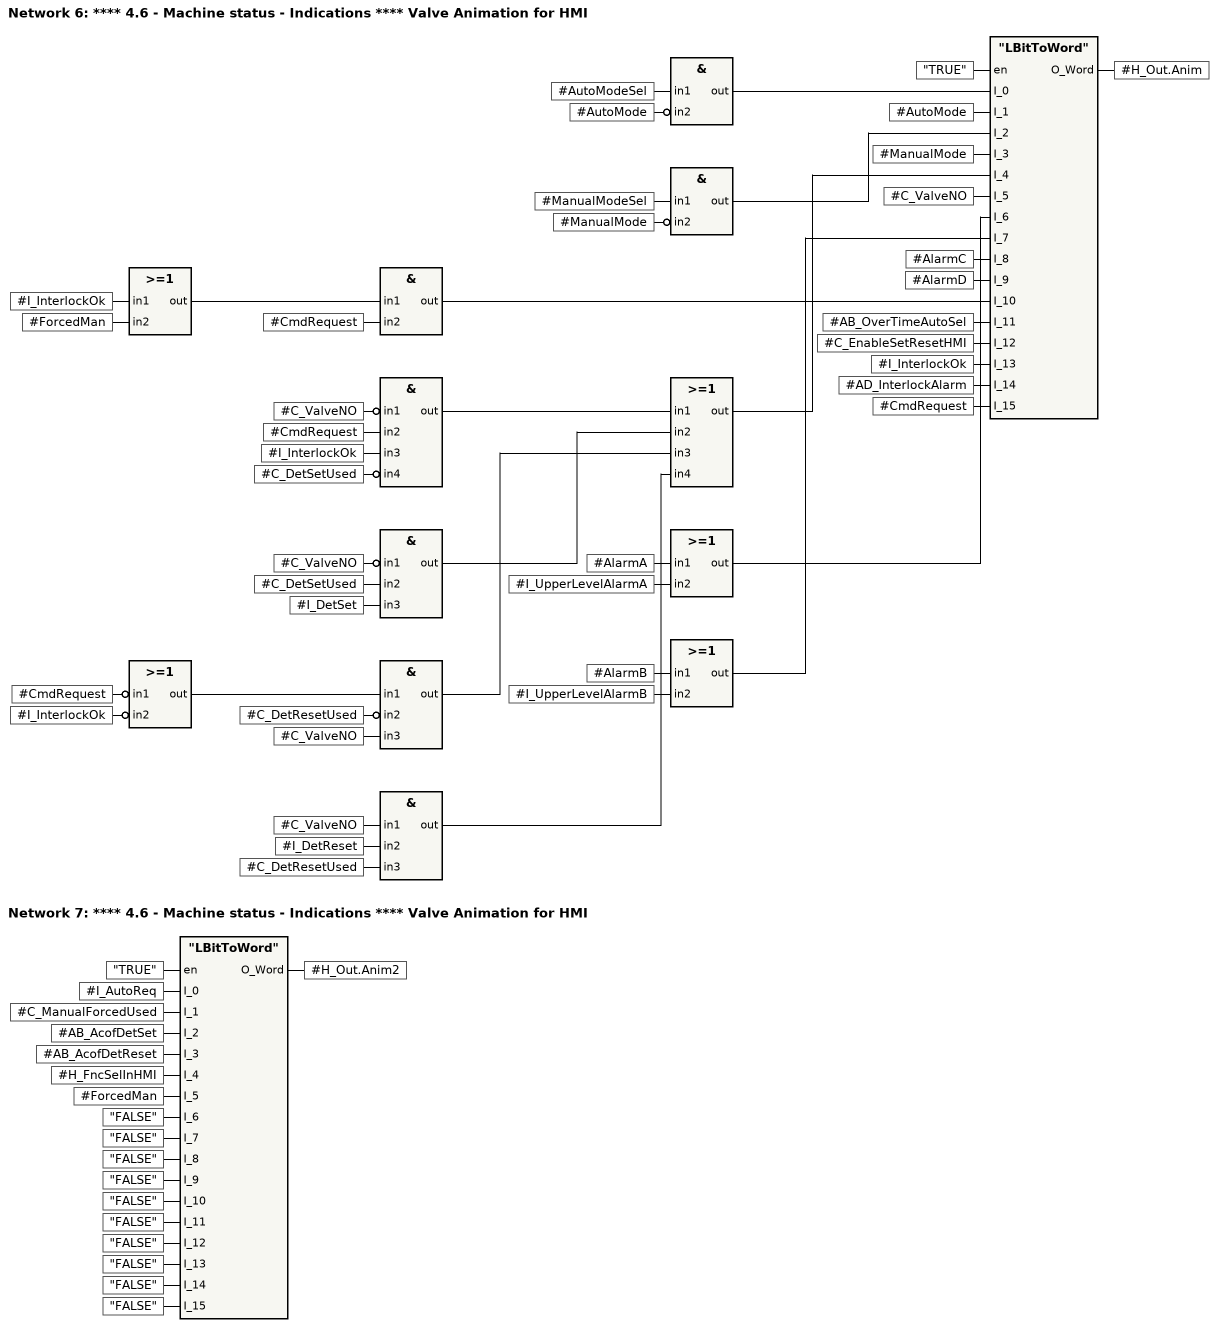
   IF "TRUE" THEN
       "LBitToWord"(I_0 := #AutoModeSel AND NOT #AutoMode,
                    I_1 := #AutoMode,
                    I_2 := #ManualModeSel AND NOT #ManualMode,
                    I_3 := #ManualMode,
                    I_4 := (NOT #C_ValveNO AND #CmdRequest AND #I_InterlockOk AND NOT #C_DetSetUsed) OR (NOT #C_ValveNO AND #C_DetSetUsed AND #I_DetSet) OR ((NOT #CmdRequest OR NOT #I_InterlockOk) AND NOT #C_DetResetUsed AND #C_ValveNO) OR (#C_ValveNO AND #I_DetReset AND #C_DetResetUsed),
                    I_5 := #C_ValveNO,
                    I_6 := #AlarmA OR #I_UpperLevelAlarmA,
                    I_7 := #AlarmB OR #I_UpperLevelAlarmB,
                    I_8 := #AlarmC,
                    I_9 := #AlarmD,
                    I_10 := (#I_InterlockOk OR #ForcedMan) AND #CmdRequest,
                    I_11 := #AB_OverTimeAutoSel,
                    I_12 := #C_EnableSetResetHMI,
                    I_13 := #I_InterlockOk,
                    I_14 := #AD_InterlockAlarm,
                    I_15 := #CmdRequest,
                    O_Word => #H_Out.Anim);
   END_IF;
END_REGION

REGION Network 7: **** 4.6 - Machine status - Indications **** Valve Animation for HMI
   // Valve Animation for HMI
   IF "TRUE" THEN
       "LBitToWord"(I_0 := #I_AutoReq,
                    I_1 := #C_ManualForcedUsed,
                    I_2 := #AB_AcofDetSet,
                    I_3 := #AB_AcofDetReset,
                    I_4 := #H_FncSelInHMI,
                    I_5 := #ForcedMan,
                    I_6 := "FALSE",
                    I_7 := "FALSE",
                    I_8 := "FALSE",
                    I_9 := "FALSE",
                    I_10 := "FALSE",
                    I_11 := "FALSE",
                    I_12 := "FALSE",
                    I_13 := "FALSE",
                    I_14 := "FALSE",
                    I_15 := "FALSE",
                    O_Word => #H_Out.Anim2);
   END_IF;
END_REGION

REGION Network 8: **** 4.6 - Machine status - Indications **** Valve Animation for HMI
   // Valve Animation for HMI
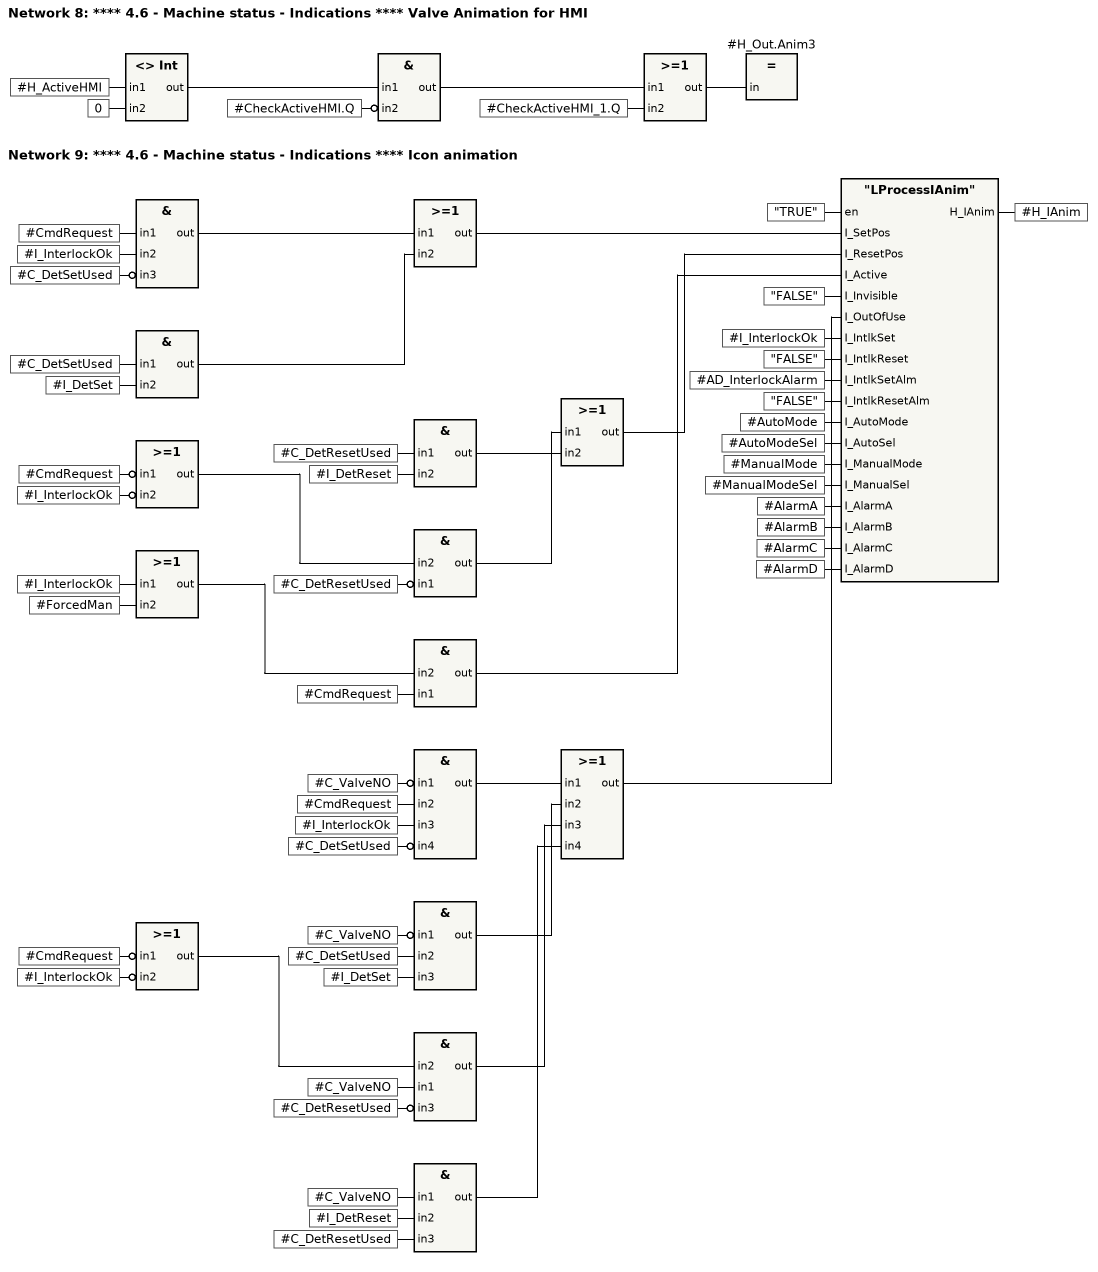
   #H_Out.Anim3 := ((#H_ActiveHMI <> 0) AND NOT #CheckActiveHMI.Q) OR #CheckActiveHMI_1.Q;
END_REGION

REGION Network 9: **** 4.6 - Machine status - Indications **** Icon animation
   // Icon animation
   IF "TRUE" THEN
       "LProcessIAnim"(I_SetPos := (#CmdRequest AND #I_InterlockOk AND NOT #C_DetSetUsed) OR (#C_DetSetUsed AND #I_DetSet),
                       I_ResetPos := ((NOT #CmdRequest OR NOT #I_InterlockOk) AND NOT #C_DetResetUsed) OR (#C_DetResetUsed AND #I_DetReset),
                       I_Active := (#I_InterlockOk OR #ForcedMan) AND #CmdRequest,
                       I_Invisible := "FALSE",
                       I_OutOfUse := (NOT #C_ValveNO AND #CmdRequest AND #I_InterlockOk AND NOT #C_DetSetUsed) OR (NOT #C_ValveNO AND #C_DetSetUsed AND #I_DetSet) OR ((NOT #CmdRequest OR NOT #I_InterlockOk) AND #C_ValveNO AND NOT #C_DetResetUsed) OR (#C_ValveNO AND #I_DetReset AND #C_DetResetUsed),
                       I_IntlkSet := #I_InterlockOk,
                       I_IntlkReset := "FALSE",
                       I_IntlkSetAlm := #AD_InterlockAlarm,
                       I_IntlkResetAlm := "FALSE",
                       I_AutoMode := #AutoMode,
                       I_AutoSel := #AutoModeSel,
                       I_ManualMode := #ManualMode,
                       I_ManualSel := #ManualModeSel,
                       I_AlarmA := #AlarmA,
                       I_AlarmB := #AlarmB,
                       I_AlarmC := #AlarmC,
                       I_AlarmD := #AlarmD,
                       H_IAnim => #H_IAnim);
   END_IF;
END_REGION

REGION Network 10: **** 4.6 - Machine status - Indications **** Valve Output animation
   // Valve Output animation
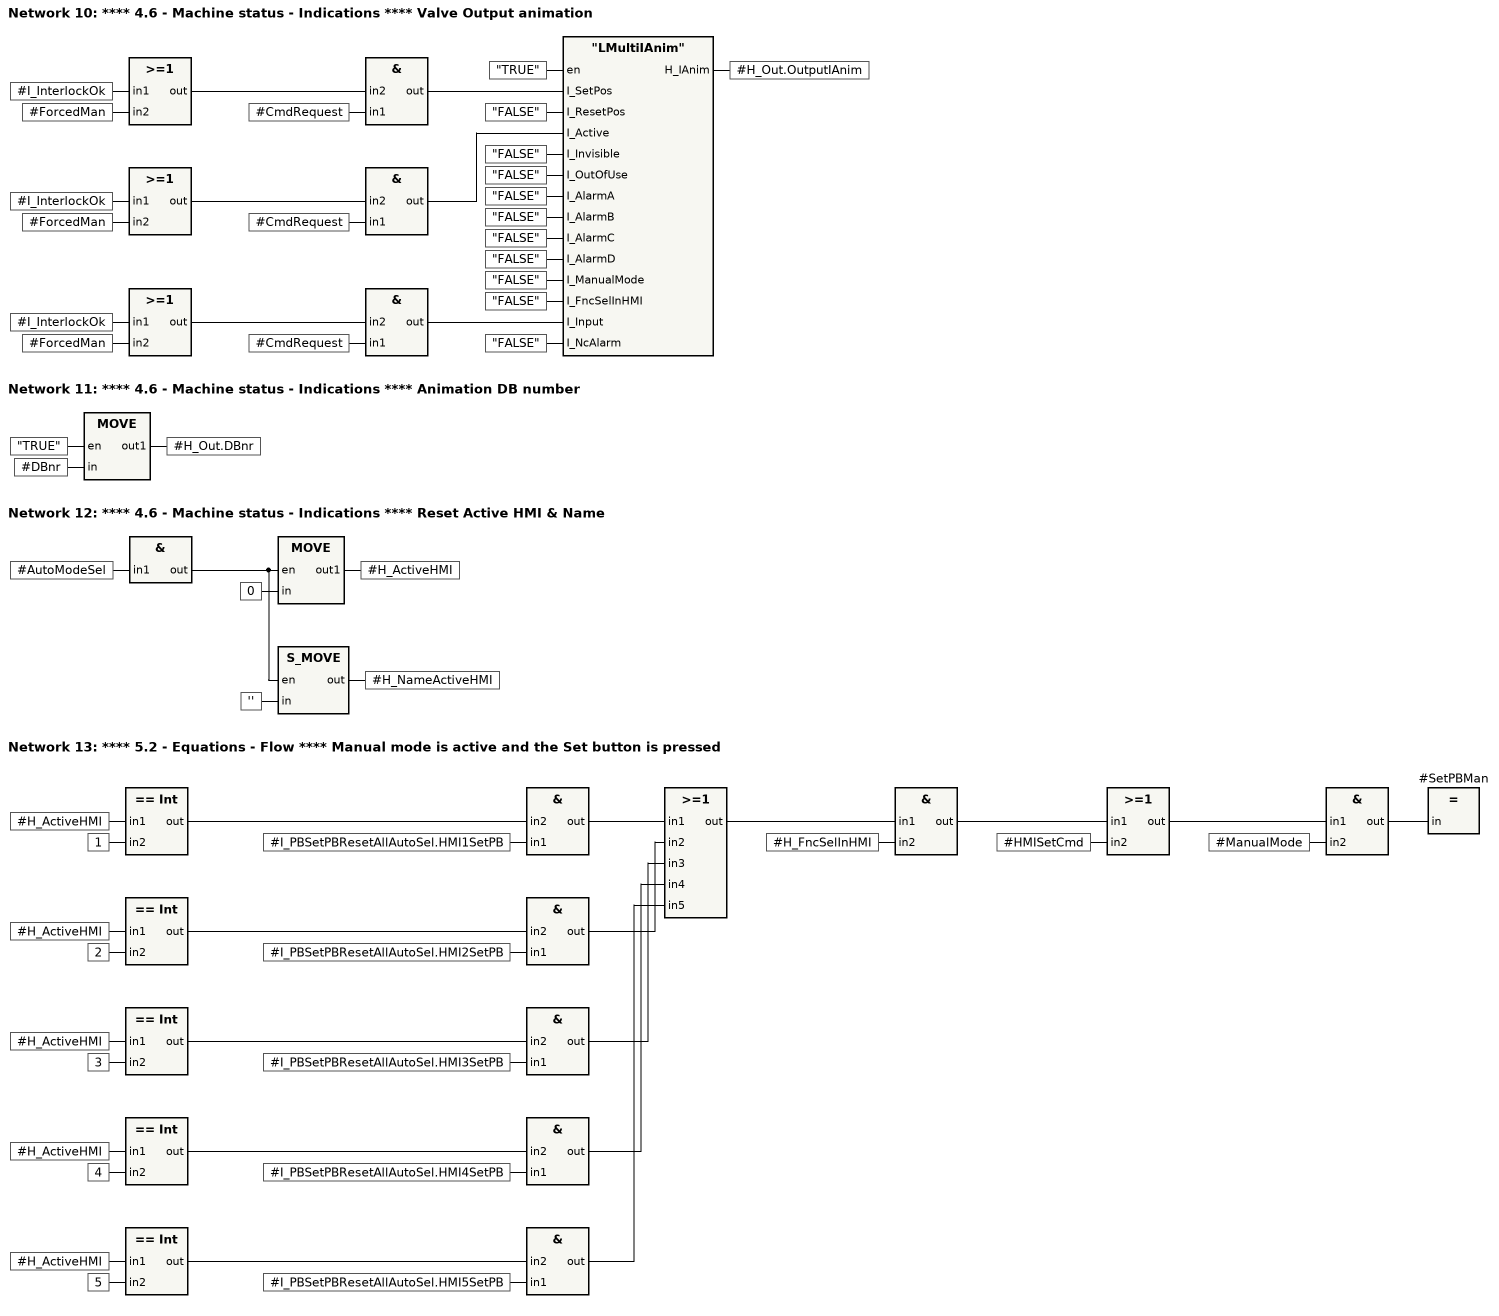
   IF "TRUE" THEN
       "LMultiIAnim"(I_SetPos := (#I_InterlockOk OR #ForcedMan) AND #CmdRequest,
                     I_ResetPos := "FALSE",
                     I_Active := (#I_InterlockOk OR #ForcedMan) AND #CmdRequest,
                     I_Invisible := "FALSE",
                     I_OutOfUse := "FALSE",
                     I_AlarmA := "FALSE",
                     I_AlarmB := "FALSE",
                     I_AlarmC := "FALSE",
                     I_AlarmD := "FALSE",
                     I_ManualMode := "FALSE",
                     I_FncSelInHMI := "FALSE",
                     I_Input := (#I_InterlockOk OR #ForcedMan) AND #CmdRequest,
                     I_NcAlarm := "FALSE",
                     H_IAnim => #H_Out.OutputIAnim);
   END_IF;
END_REGION

REGION Network 11: **** 4.6 - Machine status - Indications **** Animation DB number
   // Animation DB number
   IF "TRUE" THEN #H_Out.DBnr := #DBnr; END_IF;
END_REGION

REGION Network 12: **** 4.6 - Machine status - Indications **** Reset Active HMI & Name
   // Reset Active HMI & Name
   IF #AutoModeSel THEN
       #H_ActiveHMI := 0;
       #H_NameActiveHMI := '';
   END_IF;
END_REGION

REGION Network 13: **** 5.2 - Equations - Flow **** Manual mode is active and the Set button is pressed
   // Manual mode is active and the Set button is pressed
   #SetPBMan := (((((#H_ActiveHMI = 1) AND #I_PBSetPBResetAllAutoSel.HMI1SetPB) OR ((#H_ActiveHMI = 2) AND #I_PBSetPBResetAllAutoSel.HMI2SetPB) OR ((#H_ActiveHMI = 3) AND #I_PBSetPBResetAllAutoSel.HMI3SetPB) OR ((#H_ActiveHMI = 4) AND #I_PBSetPBResetAllAutoSel.HMI4SetPB) OR ((#H_ActiveHMI = 5) AND #I_PBSetPBResetAllAutoSel.HMI5SetPB)) AND #H_FncSelInHMI) OR #HMISetCmd) AND #ManualMode;
END_REGION

REGION Network 14: **** 5.2 - Equations - Flow **** Manual mode is active and the Reset button is pressed
   // Manual mode is active and the Reset button is pressed
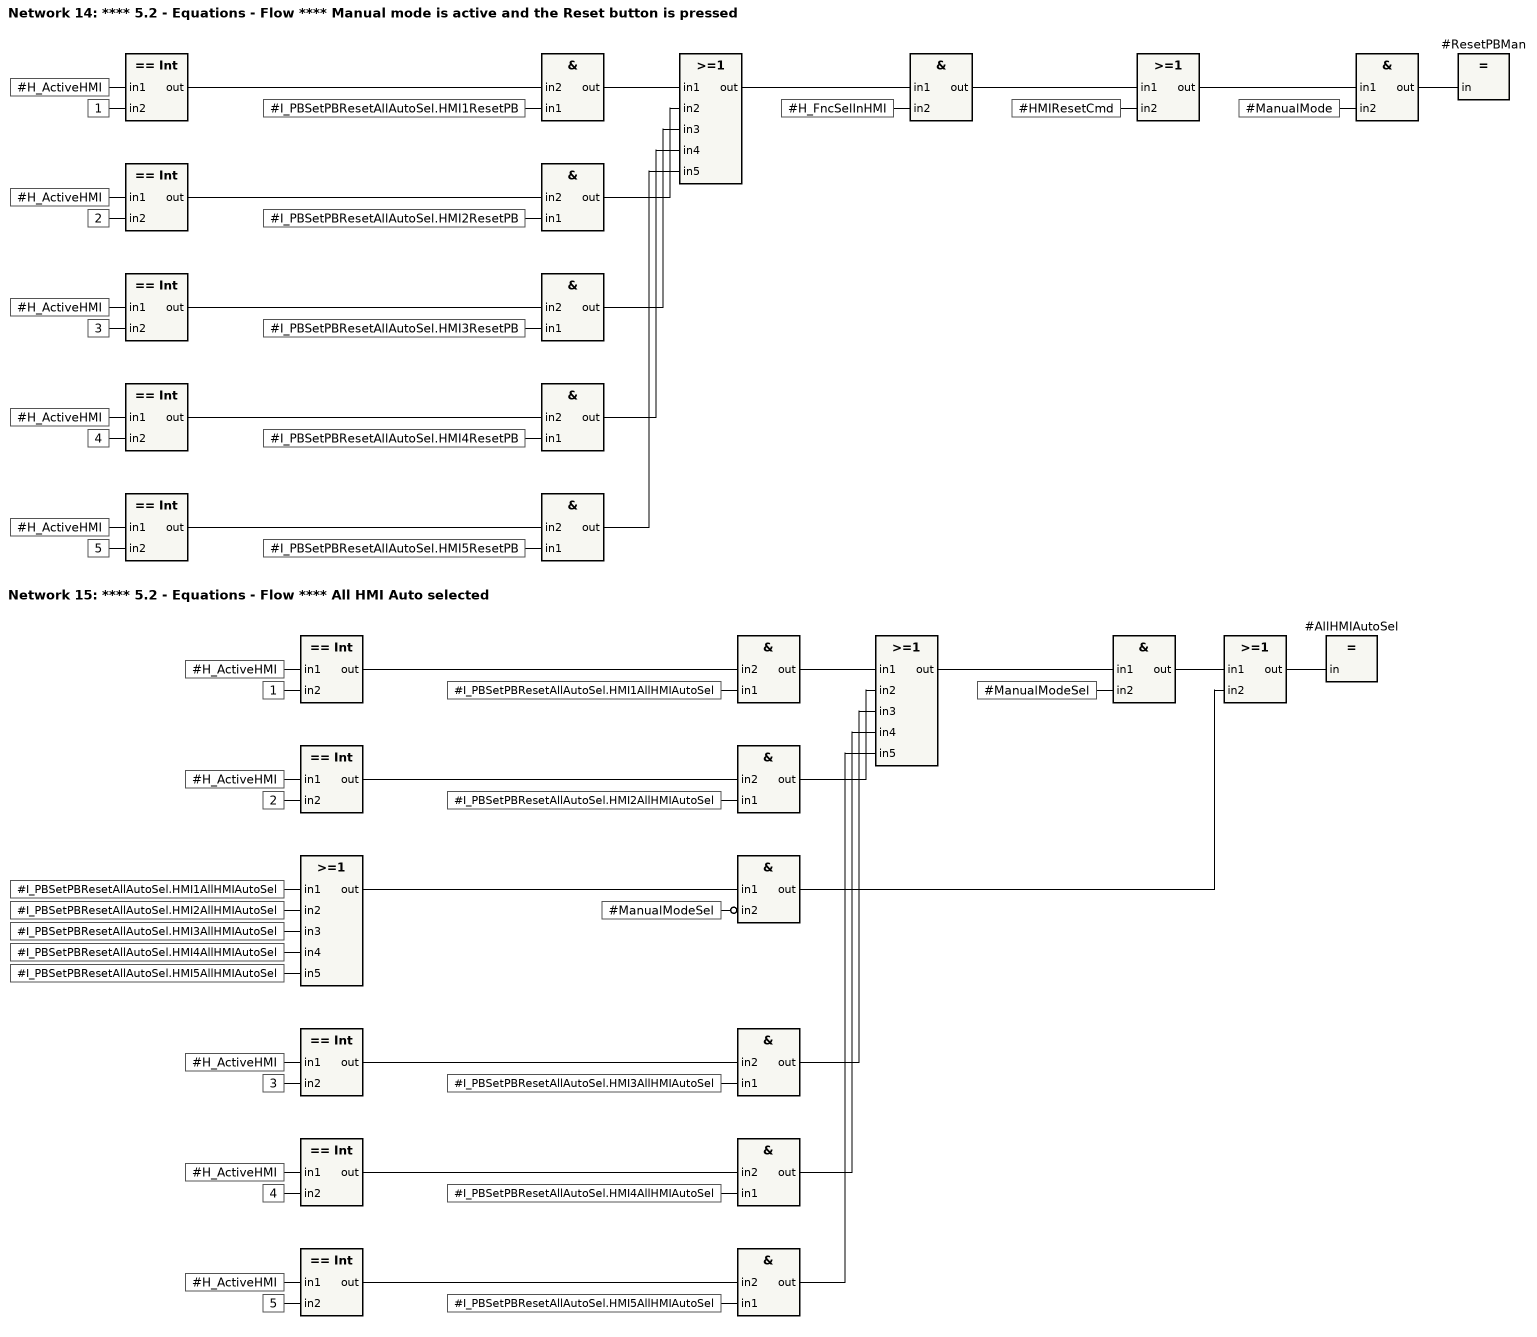
   #ResetPBMan := (((((#H_ActiveHMI = 1) AND #I_PBSetPBResetAllAutoSel.HMI1ResetPB) OR ((#H_ActiveHMI = 2) AND #I_PBSetPBResetAllAutoSel.HMI2ResetPB) OR ((#H_ActiveHMI = 3) AND #I_PBSetPBResetAllAutoSel.HMI3ResetPB) OR ((#H_ActiveHMI = 4) AND #I_PBSetPBResetAllAutoSel.HMI4ResetPB) OR ((#H_ActiveHMI = 5) AND #I_PBSetPBResetAllAutoSel.HMI5ResetPB)) AND #H_FncSelInHMI) OR #HMIResetCmd) AND #ManualMode;
END_REGION

REGION Network 15: **** 5.2 - Equations - Flow **** All HMI Auto selected
   // All HMI Auto selected
   #AllHMIAutoSel := ((((#H_ActiveHMI = 1) AND #I_PBSetPBResetAllAutoSel.HMI1AllHMIAutoSel) OR ((#H_ActiveHMI = 2) AND #I_PBSetPBResetAllAutoSel.HMI2AllHMIAutoSel) OR ((#H_ActiveHMI = 3) AND #I_PBSetPBResetAllAutoSel.HMI3AllHMIAutoSel) OR ((#H_ActiveHMI = 4) AND #I_PBSetPBResetAllAutoSel.HMI4AllHMIAutoSel) OR ((#H_ActiveHMI = 5) AND #I_PBSetPBResetAllAutoSel.HMI5AllHMIAutoSel)) AND #ManualModeSel) OR ((#I_PBSetPBResetAllAutoSel.HMI1AllHMIAutoSel OR #I_PBSetPBResetAllAutoSel.HMI2AllHMIAutoSel OR #I_PBSetPBResetAllAutoSel.HMI3AllHMIAutoSel OR #I_PBSetPBResetAllAutoSel.HMI4AllHMIAutoSel OR #I_PBSetPBResetAllAutoSel.HMI5AllHMIAutoSel) AND NOT #ManualModeSel);
END_REGION

REGION Network 16: **** 5.2 - Equations - Flow **** Check Active HMI again - HMI <> 0
   // Check Active HMI again
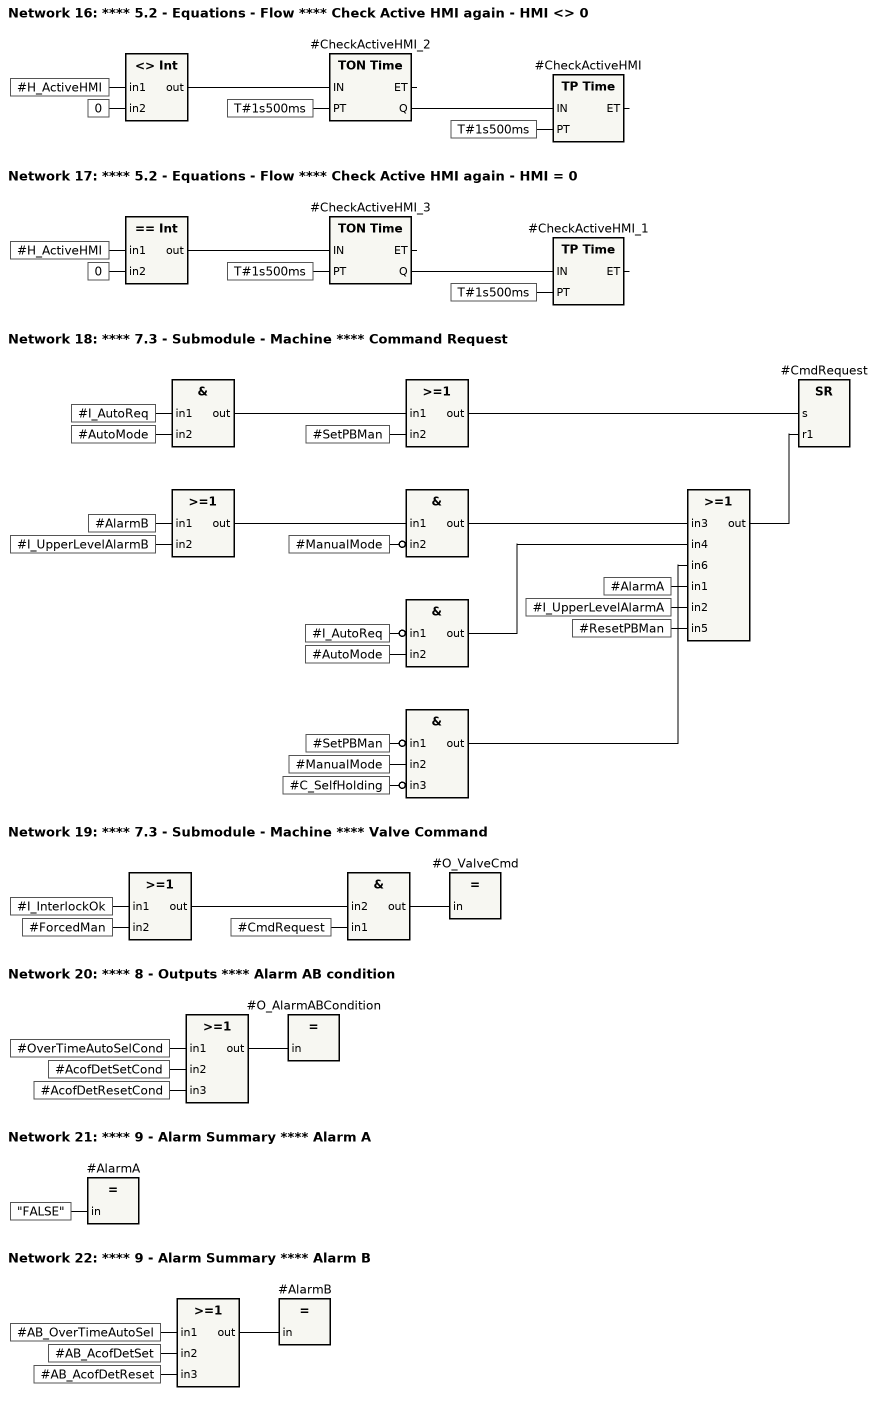
   #CheckActiveHMI_2(IN := #H_ActiveHMI <> 0, PT := T#1s500ms);   // TON
   #CheckActiveHMI(IN := #CheckActiveHMI_2.Q, PT := T#1s500ms);   // TP
END_REGION

REGION Network 17: **** 5.2 - Equations - Flow **** Check Active HMI again - HMI = 0
   // Check Active HMI again
   #CheckActiveHMI_3(IN := #H_ActiveHMI = 0, PT := T#1s500ms);   // TON
   #CheckActiveHMI_1(IN := #CheckActiveHMI_3.Q, PT := T#1s500ms);   // TP
END_REGION

REGION Network 18: **** 7.3 - Submodule - Machine **** Command Request
   // Command Request
   IF (#I_AutoReq AND #AutoMode) OR #SetPBMan THEN
       #CmdRequest := TRUE;   // SR flip-flop
   END_IF;
   IF ((#AlarmB OR #I_UpperLevelAlarmB) AND NOT #ManualMode) OR (NOT #I_AutoReq AND #AutoMode) OR (NOT #SetPBMan AND #ManualMode AND NOT #C_SelfHolding) OR #AlarmA OR #I_UpperLevelAlarmA OR #ResetPBMan THEN
       #CmdRequest := FALSE;
   END_IF;
END_REGION

REGION Network 19: **** 7.3 - Submodule - Machine **** Valve Command
   // Valve Command
   #O_ValveCmd := (#I_InterlockOk OR #ForcedMan) AND #CmdRequest;
END_REGION

REGION Network 20: **** 8 - Outputs **** Alarm AB condition
   // Alarm AB condition
   #O_AlarmABCondition := #OverTimeAutoSelCond OR #AcofDetSetCond OR #AcofDetResetCond;
END_REGION

REGION Network 21: **** 9 - Alarm Summary **** Alarm A
   // Summary of alarms A
   #AlarmA := "FALSE";
END_REGION

REGION Network 22: **** 9 - Alarm Summary **** Alarm B
   // Summary of alarms B
   #AlarmB := #AB_OverTimeAutoSel OR #AB_AcofDetSet OR #AB_AcofDetReset;
END_REGION

REGION Network 23: **** 9 - Alarm Summary **** Alarm C
   // Summary of alarms C
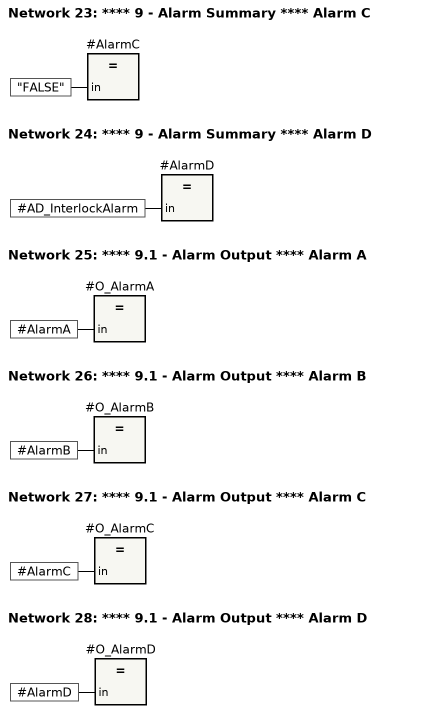
   #AlarmC := "FALSE";
END_REGION

REGION Network 24: **** 9 - Alarm Summary **** Alarm D
   // Summary of alarms D
   #AlarmD := #AD_InterlockAlarm;
END_REGION

REGION Network 25: **** 9.1 - Alarm Output **** Alarm A
   // Summary of alarms A
   #O_AlarmA := #AlarmA;
END_REGION

REGION Network 26: **** 9.1 - Alarm Output **** Alarm B
   // Summary of alarms B
   #O_AlarmB := #AlarmB;
END_REGION

REGION Network 27: **** 9.1 - Alarm Output **** Alarm C
   // Summary of alarms C
   #O_AlarmC := #AlarmC;
END_REGION

REGION Network 28: **** 9.1 - Alarm Output **** Alarm D
   // Summary of alarms D
   #O_AlarmD := #AlarmD;
END_REGION

REGION Network 29: **** 9.2 - Alarm DWord**** Alarm To DWord
   // Alarm Word
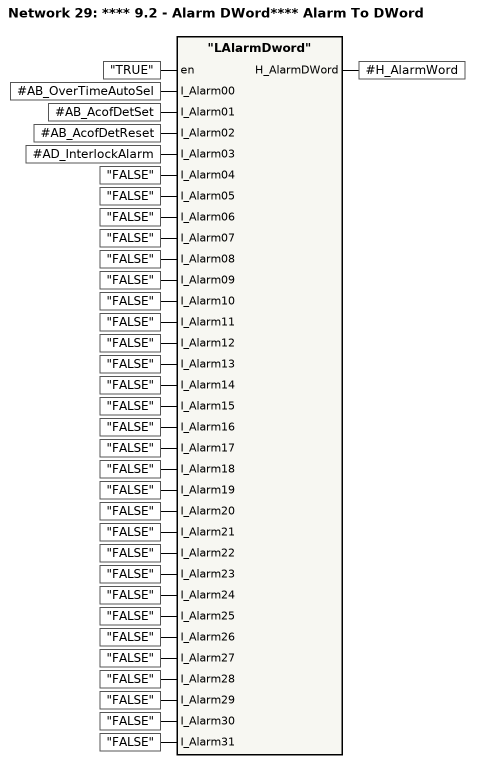
   IF "TRUE" THEN
       "LAlarmDword"(I_Alarm00 := #AB_OverTimeAutoSel,
                     I_Alarm01 := #AB_AcofDetSet,
                     I_Alarm02 := #AB_AcofDetReset,
                     I_Alarm03 := #AD_InterlockAlarm,
                     I_Alarm04 := "FALSE",
                     I_Alarm05 := "FALSE",
                     I_Alarm06 := "FALSE",
                     I_Alarm07 := "FALSE",
                     I_Alarm08 := "FALSE",
                     I_Alarm09 := "FALSE",
                     I_Alarm10 := "FALSE",
                     I_Alarm11 := "FALSE",
                     I_Alarm12 := "FALSE",
                     I_Alarm13 := "FALSE",
                     I_Alarm14 := "FALSE",
                     I_Alarm15 := "FALSE",
                     I_Alarm16 := "FALSE",
                     I_Alarm17 := "FALSE",
                     I_Alarm18 := "FALSE",
                     I_Alarm19 := "FALSE",
                     I_Alarm20 := "FALSE",
                     I_Alarm21 := "FALSE",
                     I_Alarm22 := "FALSE",
                     I_Alarm23 := "FALSE",
                     I_Alarm24 := "FALSE",
                     I_Alarm25 := "FALSE",
                     I_Alarm26 := "FALSE",
                     I_Alarm27 := "FALSE",
                     I_Alarm28 := "FALSE",
                     I_Alarm29 := "FALSE",
                     I_Alarm30 := "FALSE",
                     I_Alarm31 := "FALSE",
                     H_AlarmDWord => #H_AlarmWord);
   END_IF;
END_REGION
END_FUNCTION_BLOCK

FUNCTION_BLOCK "LProcAcofDet"   // FB1739, FBD
TITLE = LAcofDet
{ S7_Optimized_Access := 'FALSE' }
AUTHOR : VCC
FAMILY : Actuator
NAME : LAcofDet
VERSION : 1.0
// ===============================================================================
// This module handles a partdetection with all his functions and alarms
// Functions are DetCheckOn, DetCheckOff and EnableAlarm
// Outputs are DetAlarm and DetSim signal
// ===============================================================================
// stored: AutoNumber false, IsIECCheckEnabled false, SetENOAutomatically False, UDAEnableTagReadback false
   VAR_INPUT
      I_Input { ExternalAccessible := 'False'; ExternalVisible := 'False'; ExternalWritable := 'False'} : Bool;   // Actual input from sensor
      I_SignalCheckOn { ExternalAccessible := 'False'; ExternalVisible := 'False'; ExternalWritable := 'False'} : Bool;   // Signal to check signal is on
      I_SignalCheckOff { ExternalAccessible := 'False'; ExternalVisible := 'False'; ExternalWritable := 'False'} : Bool;   // Signal to check signal is off
      I_MaxAcofTime { ExternalAccessible := 'False'; ExternalVisible := 'False'; ExternalWritable := 'False'} : DInt;   // Maximum Time (ms) that the function may run (create overtime)
      I_AlarmClass { ExternalAccessible := 'False'; ExternalVisible := 'False'; ExternalWritable := 'False'} : Char;   // Alarm class -> A - B - C - D or E
      I_EnableAlarm { ExternalAccessible := 'False'; ExternalVisible := 'False'; ExternalWritable := 'False'} : Bool;   // Enable alarms
      I_Simulate { ExternalAccessible := 'False'; ExternalVisible := 'False'; ExternalWritable := 'False'} : Bool;   // Simulate modus
      I_AlarmResetPB { ExternalAccessible := 'False'; ExternalVisible := 'False'; ExternalWritable := 'False'} : Bool;   // Alarm reset pushbutton is activated
      I_Invisible { ExternalAccessible := 'False'; ExternalVisible := 'False'; ExternalWritable := 'False'} : Bool;   // Invisible
   END_VAR
   VAR_OUTPUT
      O_DetOn { ExternalAccessible := 'False'; ExternalVisible := 'False'; ExternalWritable := 'False'} : Bool;   // Detection signal to use in program
      O_Alarm { ExternalAccessible := 'False'; ExternalVisible := 'False'; ExternalWritable := 'False'} : Bool;   // Detection alarm
      O_AlarmABCondition { ExternalAccessible := 'False'; ExternalVisible := 'False'; ExternalWritable := 'False'} : Bool;   // Alarm AB condition
      O_AlarmDisabled { ExternalAccessible := 'False'; ExternalVisible := 'False'; ExternalWritable := 'False'} : Bool;   // Alarm disabled from HMI
      H_IAnim { ExternalAccessible := 'False'; ExternalVisible := 'False'; ExternalWritable := 'False'} : Word;   // For animation of the icon
   END_VAR
   VAR DB_SPECIFIC
      H_In : Struct   // HMI
         DisableAlarm : Bool;   // Disable alarm from HMI
      END_STRUCT;
      H_Out : Struct   // HMI
         Anim : Word;   // HMI Animation of the object
         DBnr : Int;   // HMI Animation DB number
      END_STRUCT;
      DetOn { ExternalAccessible := 'False'; ExternalVisible := 'False'; ExternalWritable := 'False'} : Bool;   // Static variable of O_DetOn
      DetOvtAlarm { ExternalAccessible := 'False'; ExternalVisible := 'False'; ExternalWritable := 'False'} : Bool;   // Static variable of O_DetAlarm
      Alarm { ExternalAccessible := 'False'; ExternalVisible := 'False'; ExternalWritable := 'False'} : Bool;   // Alarm condition
      AlarmClass_A { ExternalAccessible := 'False'; ExternalVisible := 'False'; ExternalWritable := 'False'} : Bool;   // The alarm is from alarm class A
      AlarmClass_B { ExternalAccessible := 'False'; ExternalVisible := 'False'; ExternalWritable := 'False'} : Bool;   // The alarm is from alarm class B
      AlarmClass_C { ExternalAccessible := 'False'; ExternalVisible := 'False'; ExternalWritable := 'False'} : Bool;   // The alarm is from alarm class C
      AlarmClass_D { ExternalAccessible := 'False'; ExternalVisible := 'False'; ExternalWritable := 'False'} : Bool;   // The alarm is from alarm class D
      AlarmClass_E { ExternalAccessible := 'False'; ExternalVisible := 'False'; ExternalWritable := 'False'} : Bool;   // The alarm is from alarm class E
      DBnr { ExternalAccessible := 'False'; ExternalVisible := 'False'; ExternalWritable := 'False'} : Int;   // HMI DB number
   END_VAR
   VAR
      MaxTimeTimer { ExternalAccessible := 'False'; ExternalVisible := 'False'; ExternalWritable := 'False'; S7_SetPoint := 'True'} : "LTimer";   // Creating alarm overtime
   END_VAR
BEGIN

NETWORK
TITLE = **** 1 - Inputs **** DB number
// DB number
      L     DINO;
      T     #DBnr;

NETWORK
TITLE = **** 1 - Inputs **** Alarm class
// Alarm class
// Alarm class = E
      L     #I_AlarmClass;
      L     'E';
      ==I;
      =     #AlarmClass_E;

// Alarm class = D
      L     #I_AlarmClass;
      L     'D';
      ==I;
      =     #AlarmClass_D;

// Alarm class = C
      L     #I_AlarmClass;
      L     'C';
      ==I;
      =     #AlarmClass_C;

// Alarm class = B
      L     #I_AlarmClass;
      L     'B';
      ==I;
      =     #AlarmClass_B;

// Alarm class = A
      AN    #AlarmClass_B;
      AN    #AlarmClass_C;
      AN    #AlarmClass_D;
      AN    #AlarmClass_E;
      =     #AlarmClass_A;


REGION Network 3: **** 2.2 - Alarms - Alarm generation **** Creating alarm overtime
   // Creating alarm overtime
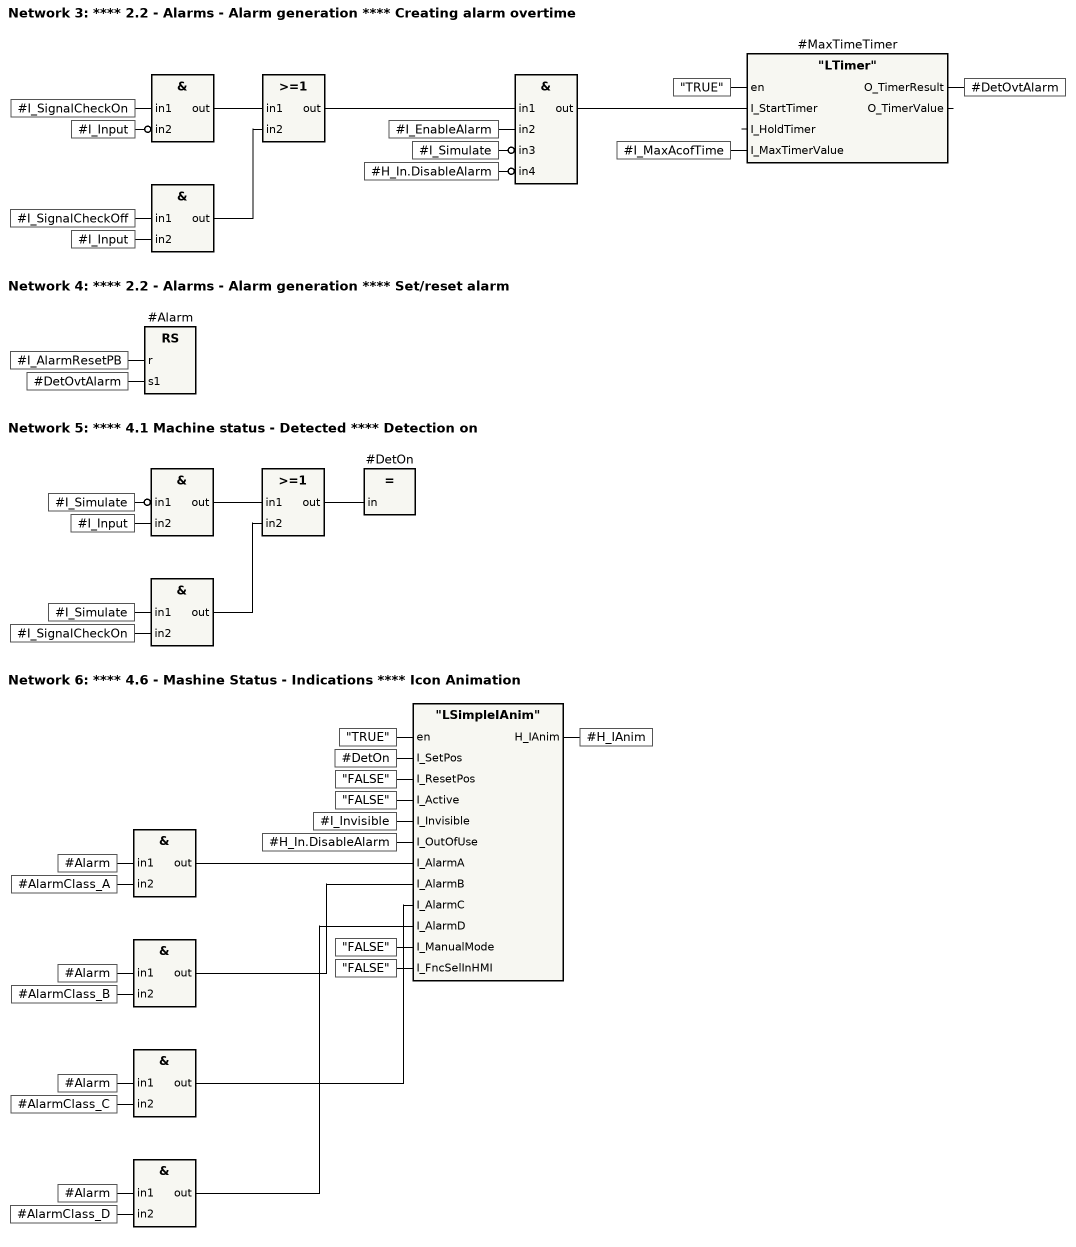
   IF "TRUE" THEN
       #MaxTimeTimer(I_StartTimer := ((#I_SignalCheckOn AND NOT #I_Input) OR (#I_SignalCheckOff AND #I_Input)) AND #I_EnableAlarm AND NOT #I_Simulate AND NOT #H_In.DisableAlarm,   // "LTimer"
                     I_MaxTimerValue := #I_MaxAcofTime,
                     O_TimerResult => #DetOvtAlarm);
   END_IF;
END_REGION

REGION Network 4: **** 2.2 - Alarms - Alarm generation **** Set/reset alarm
   // Set/reset alarm
   IF #I_AlarmResetPB THEN
       #Alarm := FALSE;   // RS flip-flop
   END_IF;
   IF #DetOvtAlarm THEN #Alarm := TRUE; END_IF;
END_REGION

REGION Network 5: **** 4.1 Machine status - Detected **** Detection on
   // Detection on
   #DetOn := (NOT #I_Simulate AND #I_Input) OR (#I_Simulate AND #I_SignalCheckOn);
END_REGION

REGION Network 6: **** 4.6 - Mashine Status - Indications **** Icon Animation
   // Icon Animation
   IF "TRUE" THEN
       "LSimpleIAnim"(I_SetPos := #DetOn,
                      I_ResetPos := "FALSE",
                      I_Active := "FALSE",
                      I_Invisible := #I_Invisible,
                      I_OutOfUse := #H_In.DisableAlarm,
                      I_AlarmA := #Alarm AND #AlarmClass_A,
                      I_AlarmB := #Alarm AND #AlarmClass_B,
                      I_AlarmC := #Alarm AND #AlarmClass_C,
                      I_AlarmD := #Alarm AND #AlarmClass_D,
                      I_ManualMode := "FALSE",
                      I_FncSelInHMI := "FALSE",
                      H_IAnim => #H_IAnim);
   END_IF;
END_REGION

REGION Network 7: **** 4.6 - Machine Status - Indications **** Animation
   // Animation
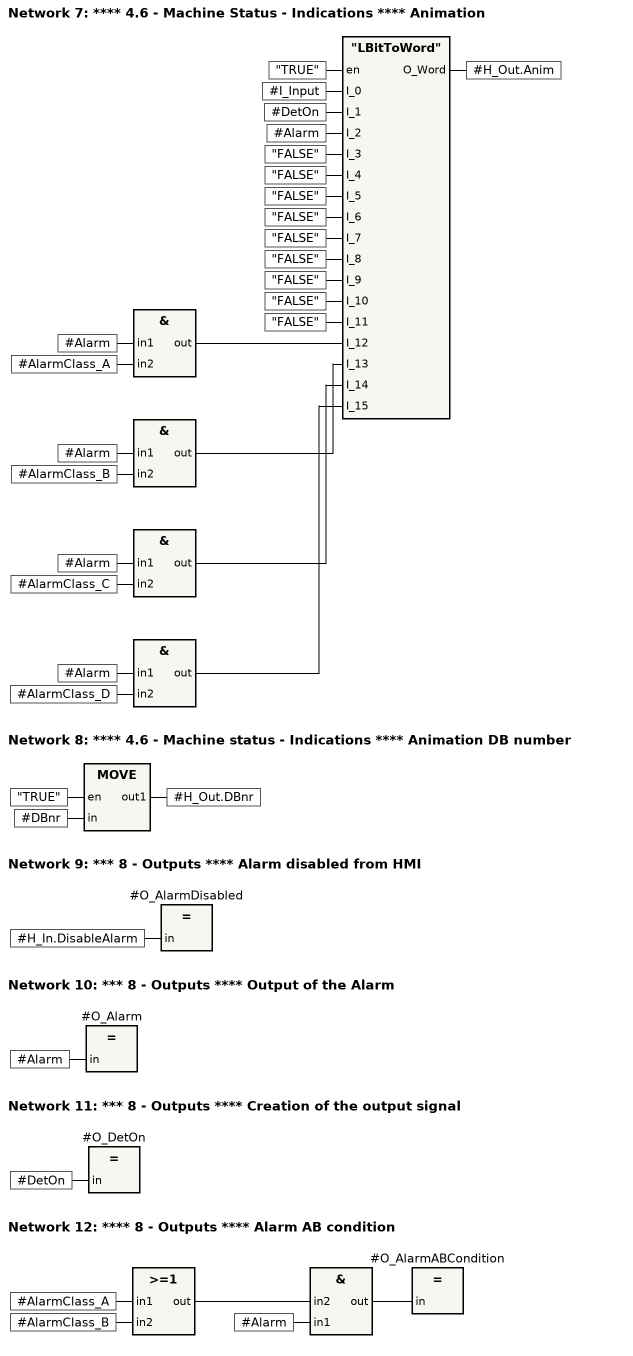
   IF "TRUE" THEN
       "LBitToWord"(I_0 := #I_Input,
                    I_1 := #DetOn,
                    I_2 := #Alarm,
                    I_3 := "FALSE",
                    I_4 := "FALSE",
                    I_5 := "FALSE",
                    I_6 := "FALSE",
                    I_7 := "FALSE",
                    I_8 := "FALSE",
                    I_9 := "FALSE",
                    I_10 := "FALSE",
                    I_11 := "FALSE",
                    I_12 := #Alarm AND #AlarmClass_A,
                    I_13 := #Alarm AND #AlarmClass_B,
                    I_14 := #Alarm AND #AlarmClass_C,
                    I_15 := #Alarm AND #AlarmClass_D,
                    O_Word => #H_Out.Anim);
   END_IF;
END_REGION

REGION Network 8: **** 4.6 - Machine status - Indications **** Animation DB number
   // Animation DB number
   IF "TRUE" THEN #H_Out.DBnr := #DBnr; END_IF;
END_REGION

REGION Network 9: *** 8 - Outputs **** Alarm disabled from HMI
   // Alarm disabled from HMI
   #O_AlarmDisabled := #H_In.DisableAlarm;
END_REGION

REGION Network 10: *** 8 - Outputs **** Output of the Alarm
   // Output of the Alarm
   #O_Alarm := #Alarm;
END_REGION

REGION Network 11: *** 8 - Outputs **** Creation of the output signal
   // Creation of the output signal
   #O_DetOn := #DetOn;
END_REGION

REGION Network 12: **** 8 - Outputs **** Alarm AB condition
   // Alarm AB condition
   #O_AlarmABCondition := (#AlarmClass_A OR #AlarmClass_B) AND #Alarm;
END_REGION
END_FUNCTION_BLOCK

FUNCTION_BLOCK "LProcObjectMode"   // FB1715, FBD
TITLE = LProcObjectMode
{ S7_Optimized_Access := 'FALSE' }
AUTHOR : VCC
FAMILY : ProcEq
NAME : LProcMod
VERSION : 0.1
// ===============================================================================
// This module handles the modes of the process equipments.
// ===============================================================================
// stored: AutoNumber false, IsIECCheckEnabled false, SetENOAutomatically False, UDAEnableTagReadback false
   VAR_INPUT
      I_StartPB { ExternalAccessible := 'False'; ExternalVisible := 'False'; ExternalWritable := 'False'} : Bool;   // Summary Start PB's
      I_EnableAlarm { ExternalAccessible := 'False'; ExternalVisible := 'False'; ExternalWritable := 'False'} : Bool;   // Enable Alarm for the Acof detections
      I_AlarmResetPB { ExternalAccessible := 'False'; ExternalVisible := 'False'; ExternalWritable := 'False'} : Bool;   // Alarm reset pushbutton is activated
      I_GeneralAutoSel { ExternalAccessible := 'False'; ExternalVisible := 'False'; ExternalWritable := 'False'} : Bool;   // General Auto Selection Request
      I_AlarmA { ExternalAccessible := 'False'; ExternalVisible := 'False'; ExternalWritable := 'False'} : Bool;   // Summation Alarm A of roller.
      I_AlarmB { ExternalAccessible := 'False'; ExternalVisible := 'False'; ExternalWritable := 'False'} : Bool;   // Summation Alarm B of roller.
      I_UpperLevelAlarmA { ExternalAccessible := 'False'; ExternalVisible := 'False'; ExternalWritable := 'False'} : Bool;   // Alarm A active from the top level
      I_UpperLevelAlarmB { ExternalAccessible := 'False'; ExternalVisible := 'False'; ExternalWritable := 'False'} : Bool;   // Alarm B active from the top level
      H_HMIModeCmd : Word;   // Mode commands from HMI
   END_VAR
   VAR_OUTPUT
      O_AutoMode { ExternalAccessible := 'False'; ExternalVisible := 'False'; ExternalWritable := 'False'} : Bool;   // Auto mode
      O_ManualMode { ExternalAccessible := 'False'; ExternalVisible := 'False'; ExternalWritable := 'False'} : Bool;   // Manual mode
      O_AutoModeSel { ExternalAccessible := 'False'; ExternalVisible := 'False'; ExternalWritable := 'False'} : Bool;   // Auto Mode Selected
      O_ManualModeSel { ExternalAccessible := 'False'; ExternalVisible := 'False'; ExternalWritable := 'False'} : Bool;   // Manual Mode Selected
      O_ForcedMan { ExternalAccessible := 'False'; ExternalVisible := 'False'; ExternalWritable := 'False'} : Bool;   // Manual Forced Active
      O_FncSelInHMI { ExternalAccessible := 'False'; ExternalVisible := 'False'; ExternalWritable := 'False'} : Bool;   // Manual Selection from HMI
      O_OverTimeAutoSelCond { ExternalAccessible := 'False'; ExternalVisible := 'False'; ExternalWritable := 'False'} : Bool;   // Overtime Auto selected condition
      O_OverTimeAutoSel { ExternalAccessible := 'False'; ExternalVisible := 'False'; ExternalWritable := 'False'} : Bool;   // Alarm Overtime Auto selected
      O_HMISetCmd { ExternalAccessible := 'False'; ExternalVisible := 'False'; ExternalWritable := 'False'} : Bool;   // Set Command on HMI
      O_HMIResetCmd { ExternalAccessible := 'False'; ExternalVisible := 'False'; ExternalWritable := 'False'} : Bool;   // Reset Command on HMI
   END_VAR
   VAR DB_SPECIFIC
      AutoMode { ExternalAccessible := 'False'; ExternalVisible := 'False'; ExternalWritable := 'False'} : Bool;   // Auto mode
      ManualMode { ExternalAccessible := 'False'; ExternalVisible := 'False'; ExternalWritable := 'False'} : Bool;   // Manual mode
      AutoModeSel { ExternalAccessible := 'False'; ExternalVisible := 'False'; ExternalWritable := 'False'} : Bool;   // Auto Mode Selected
      ManualModeSel { ExternalAccessible := 'False'; ExternalVisible := 'False'; ExternalWritable := 'False'} : Bool;   // Manual Mode Selected
      ForcedMan { ExternalAccessible := 'False'; ExternalVisible := 'False'; ExternalWritable := 'False'} : Bool;   // Forced manual active
      H_AutoModeSel { ExternalAccessible := 'False'; ExternalVisible := 'False'; ExternalWritable := 'False'} : Bool;   // Auto Mode Selection from HMI
      H_ManualModeSel { ExternalAccessible := 'False'; ExternalVisible := 'False'; ExternalWritable := 'False'} : Bool;   // Manual Mode Selection from HMI
      H_FncSelInHMI { ExternalAccessible := 'False'; ExternalVisible := 'False'; ExternalWritable := 'False'} : Bool;   // Manual selection from HMI
      H_ForcedMan { ExternalAccessible := 'False'; ExternalVisible := 'False'; ExternalWritable := 'False'} : Bool;   // Forced manual from HMI
      OvTimeAutoSel { ExternalAccessible := 'False'; ExternalVisible := 'False'; ExternalWritable := 'False'} : Bool;   // Alarm Overtime Auto selected and Component activated
      EdgeForceMan { ExternalAccessible := 'False'; ExternalVisible := 'False'; ExternalWritable := 'False'} : Bool;   // Edge Forced Manual from HMI
      ResetForcedMan { ExternalAccessible := 'False'; ExternalVisible := 'False'; ExternalWritable := 'False'} : Bool;   // Reset Forced Manual
      ForcedManTimer { ExternalAccessible := 'False'; ExternalVisible := 'False'; ExternalWritable := 'False'} : Bool;   // Forced manual timer
   END_VAR
   VAR
      TimerOvtAutoSel { ExternalAccessible := 'False'; ExternalVisible := 'False'; ExternalWritable := 'False'; S7_SetPoint := 'True'} : "LTimer";   // Timer Overtime Auto Selected
      TimerForcedMan { ExternalAccessible := 'False'; ExternalVisible := 'False'; ExternalWritable := 'False'; S7_SetPoint := 'True'} : "LTimer";   // Timer Manual Forced
      OvtAutoSel { ExternalAccessible := 'False'; ExternalVisible := 'False'; ExternalWritable := 'False'; S7_SetPoint := 'True'} : "LProc1AlarmMultiIn";   // Alarm Overtime Auto Selected
   END_VAR
   VAR_TEMP   // added for the SCL form of the ladder/FBD networks
      _w1 : Bool;
   END_VAR
BEGIN

REGION Network 1: **** 1 - Inputs **** Extract the modeselection from HMI
   // Extract the modeselection from HMI
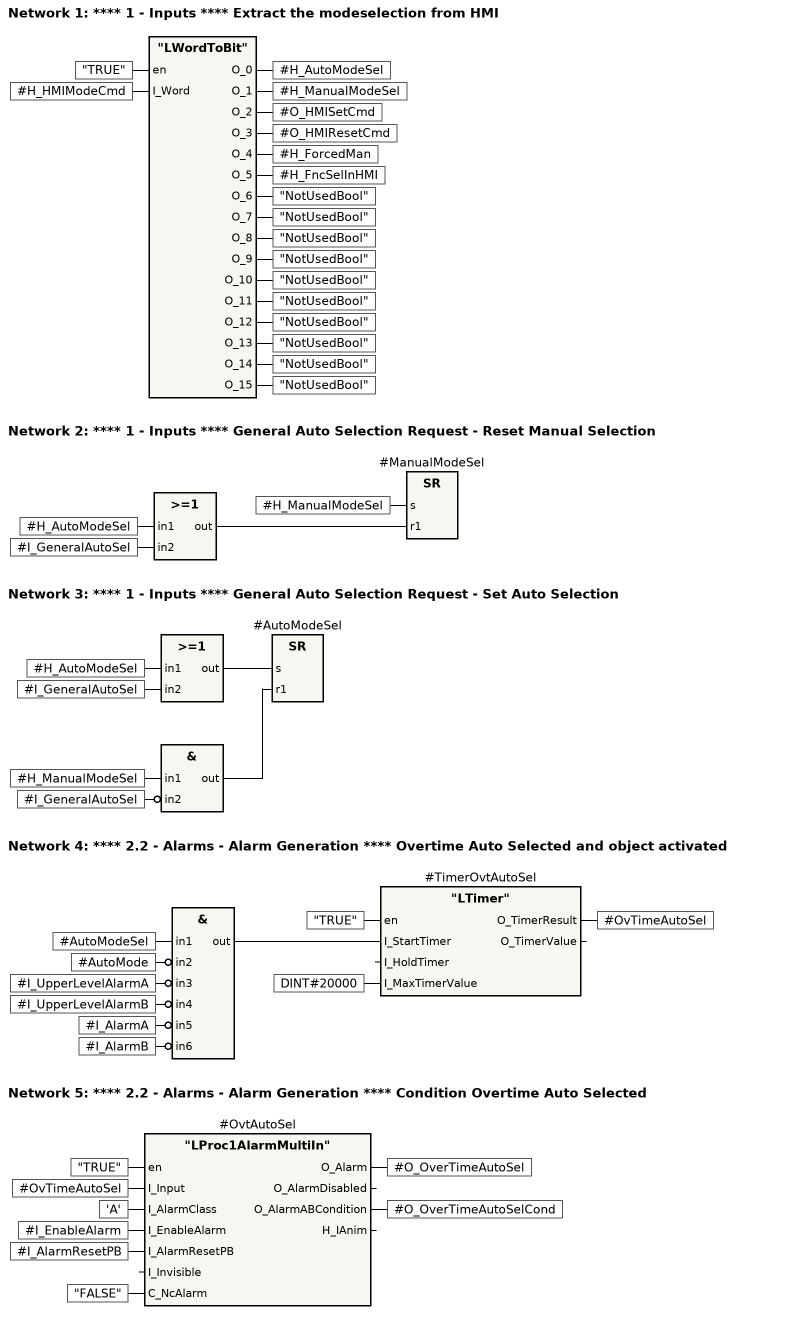
   IF "TRUE" THEN
       "LWordToBit"(I_Word := #H_HMIModeCmd,
                    O_0 => #H_AutoModeSel,
                    O_1 => #H_ManualModeSel,
                    O_2 => #O_HMISetCmd,
                    O_3 => #O_HMIResetCmd,
                    O_4 => #H_ForcedMan,
                    O_5 => #H_FncSelInHMI,
                    O_6 => "NotUsedBool",
                    O_7 => "NotUsedBool",
                    O_8 => "NotUsedBool",
                    O_9 => "NotUsedBool",
                    O_10 => "NotUsedBool",
                    O_11 => "NotUsedBool",
                    O_12 => "NotUsedBool",
                    O_13 => "NotUsedBool",
                    O_14 => "NotUsedBool",
                    O_15 => "NotUsedBool");
   END_IF;
END_REGION

REGION Network 2: **** 1 - Inputs **** General Auto Selection Request - Reset Manual Selection
   // General Auto Selection Request - Reset Manual Selection
   IF #H_ManualModeSel THEN
       #ManualModeSel := TRUE;   // SR flip-flop
   END_IF;
   IF #H_AutoModeSel OR #I_GeneralAutoSel THEN #ManualModeSel := FALSE; END_IF;
END_REGION

REGION Network 3: **** 1 - Inputs **** General Auto Selection Request - Set Auto Selection
   // General Auto Selection Request - Set Auto Selection
   IF #H_AutoModeSel OR #I_GeneralAutoSel THEN
       #AutoModeSel := TRUE;   // SR flip-flop
   END_IF;
   IF #H_ManualModeSel AND NOT #I_GeneralAutoSel THEN #AutoModeSel := FALSE; END_IF;
END_REGION

REGION Network 4: **** 2.2 - Alarms - Alarm Generation **** Overtime Auto Selected and object activated
   // Overtime Auto Selected and object activated
   IF "TRUE" THEN
       #TimerOvtAutoSel(I_StartTimer := #AutoModeSel AND NOT #AutoMode AND NOT #I_UpperLevelAlarmA AND NOT #I_UpperLevelAlarmB AND NOT #I_AlarmA AND NOT #I_AlarmB,   // "LTimer"
                        I_MaxTimerValue := DINT#20000,
                        O_TimerResult => #OvTimeAutoSel);
   END_IF;
END_REGION

REGION Network 5: **** 2.2 - Alarms - Alarm Generation **** Condition Overtime Auto Selected
   // Condition Overtime Auto Selected
   IF "TRUE" THEN
       #OvtAutoSel(I_Input := #OvTimeAutoSel,   // "LProc1AlarmMultiIn"
                   I_AlarmClass := 'A',
                   I_EnableAlarm := #I_EnableAlarm,
                   I_AlarmResetPB := #I_AlarmResetPB,
                   C_NcAlarm := "FALSE",
                   O_Alarm => #O_OverTimeAutoSel,
                   O_AlarmABCondition => #O_OverTimeAutoSelCond);
   END_IF;
END_REGION

REGION Network 6: **** 4.5 - Machine Status - Modes **** Auto mode
   // Auto mode
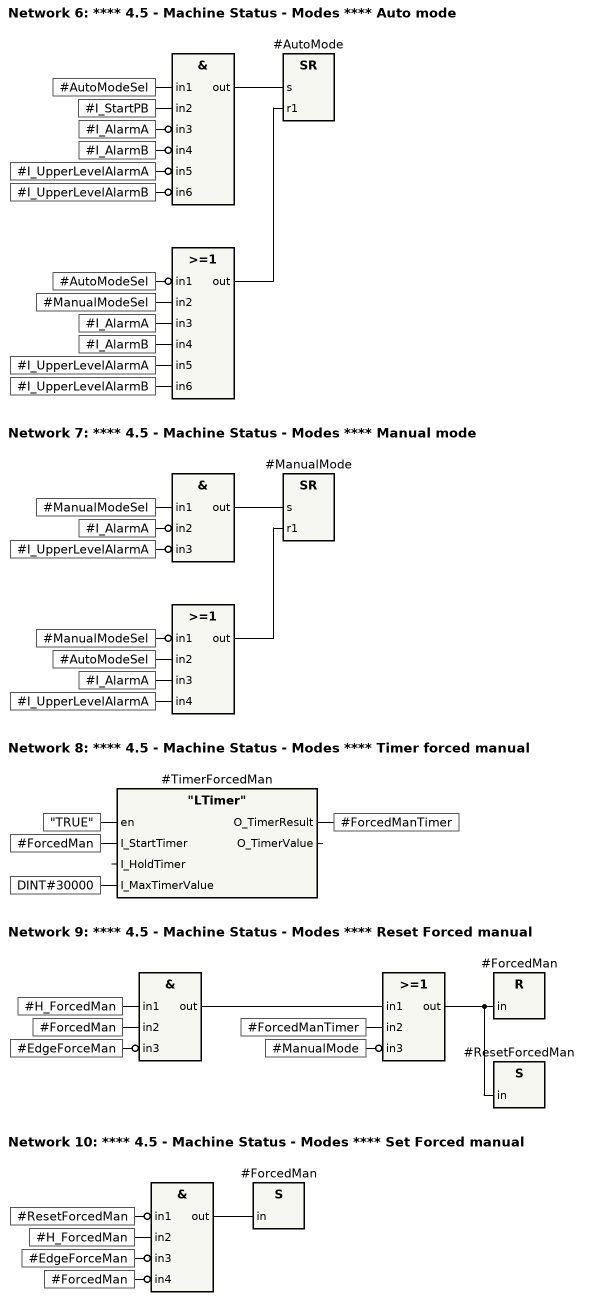
   IF #AutoModeSel AND #I_StartPB AND NOT #I_AlarmA AND NOT #I_AlarmB AND NOT #I_UpperLevelAlarmA AND NOT #I_UpperLevelAlarmB THEN
       #AutoMode := TRUE;   // SR flip-flop
   END_IF;
   IF NOT #AutoModeSel OR #ManualModeSel OR #I_AlarmA OR #I_AlarmB OR #I_UpperLevelAlarmA OR #I_UpperLevelAlarmB THEN
       #AutoMode := FALSE;
   END_IF;
END_REGION

REGION Network 7: **** 4.5 - Machine Status - Modes **** Manual mode
   // Manual mode
   IF #ManualModeSel AND NOT #I_AlarmA AND NOT #I_UpperLevelAlarmA THEN
       #ManualMode := TRUE;   // SR flip-flop
   END_IF;
   IF NOT #ManualModeSel OR #AutoModeSel OR #I_AlarmA OR #I_UpperLevelAlarmA THEN
       #ManualMode := FALSE;
   END_IF;
END_REGION

REGION Network 8: **** 4.5 - Machine Status - Modes **** Timer forced manual
   // Timer forced manual
   IF "TRUE" THEN
       #TimerForcedMan(I_StartTimer := #ForcedMan, I_MaxTimerValue := DINT#30000, O_TimerResult => #ForcedManTimer);   // "LTimer"
   END_IF;
END_REGION

REGION Network 9: **** 4.5 - Machine Status - Modes **** Reset Forced manual
   // Reset Forced manual
   #_w1 := (#H_ForcedMan AND #ForcedMan AND NOT #EdgeForceMan) OR #ForcedManTimer OR NOT #ManualMode;
   IF #_w1 THEN
       #ForcedMan := FALSE;
       #ResetForcedMan := TRUE;
   END_IF;
END_REGION

REGION Network 10: **** 4.5 - Machine Status - Modes **** Set Forced manual
   // Set Forced manual
   IF NOT #ResetForcedMan AND #H_ForcedMan AND NOT #EdgeForceMan AND NOT #ForcedMan THEN
       #ForcedMan := TRUE;
   END_IF;
END_REGION

REGION Network 11: **** 4.5 - Machine Status - Modes **** Set Forced manual
   // Set Forced manual
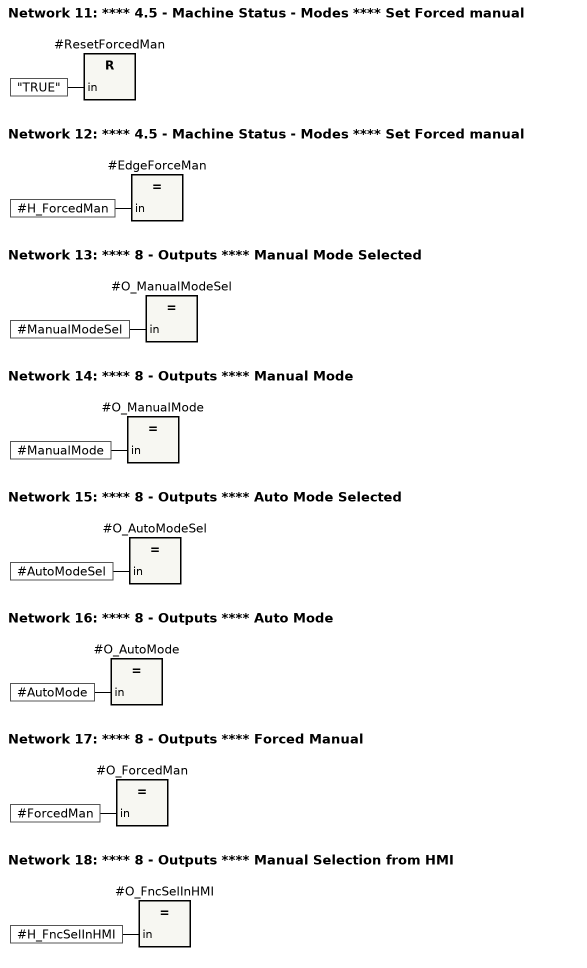
   IF "TRUE" THEN #ResetForcedMan := FALSE; END_IF;
END_REGION

REGION Network 12: **** 4.5 - Machine Status - Modes **** Set Forced manual
   // Set Forced manual
   #EdgeForceMan := #H_ForcedMan;
END_REGION

REGION Network 13: **** 8 - Outputs **** Manual Mode Selected
   // Manual Mode Selected
   #O_ManualModeSel := #ManualModeSel;
END_REGION

REGION Network 14: **** 8 - Outputs **** Manual Mode
   // Manual Mode
   #O_ManualMode := #ManualMode;
END_REGION

REGION Network 15: **** 8 - Outputs **** Auto Mode Selected
   // Auto Mode Selected
   #O_AutoModeSel := #AutoModeSel;
END_REGION

REGION Network 16: **** 8 - Outputs **** Auto Mode
   // Auto Mode
   #O_AutoMode := #AutoMode;
END_REGION

REGION Network 17: **** 8 - Outputs **** Forced Manual
   // Forced Manual
   #O_ForcedMan := #ForcedMan;
END_REGION

REGION Network 18: **** 8 - Outputs **** Manual Selection from HMI
   // Manual Selection from HMI
   #O_FncSelInHMI := #H_FncSelInHMI;
END_REGION
END_FUNCTION_BLOCK

FUNCTION_BLOCK "LProcModesSum"   // FB1702, FBD
TITLE = LProcModesSum
{ S7_Optimized_Access := 'FALSE' }
AUTHOR : VCC
FAMILY : ProcEqp
NAME : ModesSum
VERSION : 1.0
// ================================================================================
// Create the Modes Summary for 20 possible components
// ================================================================================
// stored: AutoNumber false, IsIECCheckEnabled false, SetENOAutomatically False, UDAEnableTagReadback false
   VAR_INPUT
      I_StartPB { ExternalAccessible := 'False'; ExternalVisible := 'False'; ExternalWritable := 'False'} : Bool;   // Summary of Start buttons
      I_AlarmResetPB { ExternalAccessible := 'False'; ExternalVisible := 'False'; ExternalWritable := 'False'} : Bool;   // Summary of Alarm reset buttons
      I_SafetyNotOk { ExternalAccessible := 'False'; ExternalVisible := 'False'; ExternalWritable := 'False'} : Bool;   // Safety is not ok
      I_ObjectMode1 { ExternalAccessible := 'False'; ExternalVisible := 'False'; ExternalWritable := 'False'} : Word;   // Modes Component 1
      I_ObjectMode2 { ExternalAccessible := 'False'; ExternalVisible := 'False'; ExternalWritable := 'False'} : Word;   // Modes Component 2
      I_ObjectMode3 { ExternalAccessible := 'False'; ExternalVisible := 'False'; ExternalWritable := 'False'} : Word;   // Modes Component 3
      I_ObjectMode3Used { ExternalAccessible := 'False'; ExternalVisible := 'False'; ExternalWritable := 'False'} : Bool;   // True if used
      I_ObjectMode4 { ExternalAccessible := 'False'; ExternalVisible := 'False'; ExternalWritable := 'False'} : Word;   // Modes Component 4
      I_ObjectMode4Used { ExternalAccessible := 'False'; ExternalVisible := 'False'; ExternalWritable := 'False'} : Bool;   // True if used
      I_ObjectMode5 { ExternalAccessible := 'False'; ExternalVisible := 'False'; ExternalWritable := 'False'} : Word;   // Modes Component 5
      I_ObjectMode5Used { ExternalAccessible := 'False'; ExternalVisible := 'False'; ExternalWritable := 'False'} : Bool;   // True if used
      I_ObjectMode6 { ExternalAccessible := 'False'; ExternalVisible := 'False'; ExternalWritable := 'False'} : Word;   // Modes Component 6
      I_ObjectMode6Used { ExternalAccessible := 'False'; ExternalVisible := 'False'; ExternalWritable := 'False'} : Bool;   // True if used
      I_ObjectMode7 { ExternalAccessible := 'False'; ExternalVisible := 'False'; ExternalWritable := 'False'} : Word;   // Modes Component 7
      I_ObjectMode7Used { ExternalAccessible := 'False'; ExternalVisible := 'False'; ExternalWritable := 'False'} : Bool;   // True if used
      I_ObjectMode8 { ExternalAccessible := 'False'; ExternalVisible := 'False'; ExternalWritable := 'False'} : Word;   // Modes Component 8
      I_ObjectMode8Used { ExternalAccessible := 'False'; ExternalVisible := 'False'; ExternalWritable := 'False'} : Bool;   // True if used
      I_ObjectMode9 { ExternalAccessible := 'False'; ExternalVisible := 'False'; ExternalWritable := 'False'} : Word;   // Modes Component 9
      I_ObjectMode9Used { ExternalAccessible := 'False'; ExternalVisible := 'False'; ExternalWritable := 'False'} : Bool;   // True if used
      I_ObjectMode10 { ExternalAccessible := 'False'; ExternalVisible := 'False'; ExternalWritable := 'False'} : Word;   // Modes Component 10
      I_ObjectMode10Used { ExternalAccessible := 'False'; ExternalVisible := 'False'; ExternalWritable := 'False'} : Bool;   // True if used
      I_ObjectMode11 { ExternalAccessible := 'False'; ExternalVisible := 'False'; ExternalWritable := 'False'} : Word;   // Modes Component 11
      I_ObjectMode11Used { ExternalAccessible := 'False'; ExternalVisible := 'False'; ExternalWritable := 'False'} : Bool;   // True if used
      I_ObjectMode12 { ExternalAccessible := 'False'; ExternalVisible := 'False'; ExternalWritable := 'False'} : Word;   // Modes Component 12
      I_ObjectMode12Used { ExternalAccessible := 'False'; ExternalVisible := 'False'; ExternalWritable := 'False'} : Bool;   // True if used
      I_ObjectMode13 { ExternalAccessible := 'False'; ExternalVisible := 'False'; ExternalWritable := 'False'} : Word;   // Modes Component 13
      I_ObjectMode13Used { ExternalAccessible := 'False'; ExternalVisible := 'False'; ExternalWritable := 'False'} : Bool;   // True if used
      I_ObjectMode14 { ExternalAccessible := 'False'; ExternalVisible := 'False'; ExternalWritable := 'False'} : Word;   // Modes Component 14
      I_ObjectMode14Used { ExternalAccessible := 'False'; ExternalVisible := 'False'; ExternalWritable := 'False'} : Bool;   // True if used
      I_ObjectMode15 { ExternalAccessible := 'False'; ExternalVisible := 'False'; ExternalWritable := 'False'} : Word;   // Modes Component 15
      I_ObjectMode15Used { ExternalAccessible := 'False'; ExternalVisible := 'False'; ExternalWritable := 'False'} : Bool;   // True if used
      I_ObjectMode16 { ExternalAccessible := 'False'; ExternalVisible := 'False'; ExternalWritable := 'False'} : Word;   // Modes Component 16
      I_ObjectMode16Used { ExternalAccessible := 'False'; ExternalVisible := 'False'; ExternalWritable := 'False'} : Bool;   // True if used
      I_ObjectMode17 { ExternalAccessible := 'False'; ExternalVisible := 'False'; ExternalWritable := 'False'} : Word;   // Modes Component 17
      I_ObjectMode17Used { ExternalAccessible := 'False'; ExternalVisible := 'False'; ExternalWritable := 'False'} : Bool;   // True if used
      I_ObjectMode18 { ExternalAccessible := 'False'; ExternalVisible := 'False'; ExternalWritable := 'False'} : Word;   // Modes Component 18
      I_ObjectMode18Used { ExternalAccessible := 'False'; ExternalVisible := 'False'; ExternalWritable := 'False'} : Bool;   // True if used
      I_ObjectMode19 { ExternalAccessible := 'False'; ExternalVisible := 'False'; ExternalWritable := 'False'} : Word;   // Modes Component 19
      I_ObjectMode19Used { ExternalAccessible := 'False'; ExternalVisible := 'False'; ExternalWritable := 'False'} : Bool;   // True if used
      I_ObjectMode20 { ExternalAccessible := 'False'; ExternalVisible := 'False'; ExternalWritable := 'False'} : Word;   // Modes Component 20
      I_ObjectMode20Used { ExternalAccessible := 'False'; ExternalVisible := 'False'; ExternalWritable := 'False'} : Bool;   // True if used
   END_VAR
   VAR_OUTPUT
      O_AutoSel { ExternalAccessible := 'False'; ExternalVisible := 'False'; ExternalWritable := 'False'} : Bool;   // At least one component is in auto selected
      O_Auto { ExternalAccessible := 'False'; ExternalVisible := 'False'; ExternalWritable := 'False'} : Bool;   // All the components are in auto
      O_ManSel { ExternalAccessible := 'False'; ExternalVisible := 'False'; ExternalWritable := 'False'} : Bool;   // At least one component is in manual selected
      O_Man { ExternalAccessible := 'False'; ExternalVisible := 'False'; ExternalWritable := 'False'} : Bool;   // At least one component is in manual
      O_AlarmResetPB { ExternalAccessible := 'False'; ExternalVisible := 'False'; ExternalWritable := 'False'} : Bool;   // Alarm reset button is activated
   END_VAR
   VAR DB_SPECIFIC
      H_Anim : Word;   // Mode Animation Word
      H_Anim2 : Word;   // Mode Animation Word
      H_ConfigBtnResetTM : Bool;   // From the HMI - Config internal tag
      H_ConfigBtnResetSeq : Bool;   // From the HMI - Config internal tag
      H_ModeChanged : Bool;   // From the HMI - Mode changed to Auto
      H_ScreenChanged : Bool;   // From the HMI - The screen has changed
      AutoSel1 { ExternalAccessible := 'False'; ExternalVisible := 'False'; ExternalWritable := 'False'} : Bool;   // Auto selected Component 1
      Auto1 { ExternalAccessible := 'False'; ExternalVisible := 'False'; ExternalWritable := 'False'} : Bool;   // Auto Component 1
      ManSel1 { ExternalAccessible := 'False'; ExternalVisible := 'False'; ExternalWritable := 'False'} : Bool;   // Manu selected Component 1
      Man1 { ExternalAccessible := 'False'; ExternalVisible := 'False'; ExternalWritable := 'False'} : Bool;   // Manu Component 1
      AutoSel2 { ExternalAccessible := 'False'; ExternalVisible := 'False'; ExternalWritable := 'False'} : Bool;   // Auto selected Component 2
      Auto2 { ExternalAccessible := 'False'; ExternalVisible := 'False'; ExternalWritable := 'False'} : Bool;   // Auto Component 2
      ManSel2 { ExternalAccessible := 'False'; ExternalVisible := 'False'; ExternalWritable := 'False'} : Bool;   // Manu selected Component 2
      Man2 { ExternalAccessible := 'False'; ExternalVisible := 'False'; ExternalWritable := 'False'} : Bool;   // Manu Component 2
      AutoSel3 { ExternalAccessible := 'False'; ExternalVisible := 'False'; ExternalWritable := 'False'} : Bool;   // Auto selected Component 3
      Auto3 { ExternalAccessible := 'False'; ExternalVisible := 'False'; ExternalWritable := 'False'} : Bool;   // Auto Component 3
      ManSel3 { ExternalAccessible := 'False'; ExternalVisible := 'False'; ExternalWritable := 'False'} : Bool;   // Manu selected Component 3
      Man3 { ExternalAccessible := 'False'; ExternalVisible := 'False'; ExternalWritable := 'False'} : Bool;   // Manu Component 3
      AutoSel4 { ExternalAccessible := 'False'; ExternalVisible := 'False'; ExternalWritable := 'False'} : Bool;   // Auto selected Component 4
      Auto4 { ExternalAccessible := 'False'; ExternalVisible := 'False'; ExternalWritable := 'False'} : Bool;   // Auto Component 4
      ManSel4 { ExternalAccessible := 'False'; ExternalVisible := 'False'; ExternalWritable := 'False'} : Bool;   // Manu selected Component 4
      Man4 { ExternalAccessible := 'False'; ExternalVisible := 'False'; ExternalWritable := 'False'} : Bool;   // Manu Component 4
      AutoSel5 { ExternalAccessible := 'False'; ExternalVisible := 'False'; ExternalWritable := 'False'} : Bool;   // Auto selected Component 5
      Auto5 { ExternalAccessible := 'False'; ExternalVisible := 'False'; ExternalWritable := 'False'} : Bool;   // Auto Component 5
      ManSel5 { ExternalAccessible := 'False'; ExternalVisible := 'False'; ExternalWritable := 'False'} : Bool;   // Manu selected Component 5
      Man5 { ExternalAccessible := 'False'; ExternalVisible := 'False'; ExternalWritable := 'False'} : Bool;   // Manu Component 5
      AutoSel6 { ExternalAccessible := 'False'; ExternalVisible := 'False'; ExternalWritable := 'False'} : Bool;   // Auto selected Component 6
      Auto6 { ExternalAccessible := 'False'; ExternalVisible := 'False'; ExternalWritable := 'False'} : Bool;   // Auto Component 6
      ManSel6 { ExternalAccessible := 'False'; ExternalVisible := 'False'; ExternalWritable := 'False'} : Bool;   // Manu selected Component 6
      Man6 { ExternalAccessible := 'False'; ExternalVisible := 'False'; ExternalWritable := 'False'} : Bool;   // Manu Component 6
      AutoSel7 { ExternalAccessible := 'False'; ExternalVisible := 'False'; ExternalWritable := 'False'} : Bool;   // Auto selected Component 7
      Auto7 { ExternalAccessible := 'False'; ExternalVisible := 'False'; ExternalWritable := 'False'} : Bool;   // Auto Component 7
      ManSel7 { ExternalAccessible := 'False'; ExternalVisible := 'False'; ExternalWritable := 'False'} : Bool;   // Manu selected Component 7
      Man7 { ExternalAccessible := 'False'; ExternalVisible := 'False'; ExternalWritable := 'False'} : Bool;   // Manu Component 7
      AutoSel8 { ExternalAccessible := 'False'; ExternalVisible := 'False'; ExternalWritable := 'False'} : Bool;   // Auto selected Component 8
      Auto8 { ExternalAccessible := 'False'; ExternalVisible := 'False'; ExternalWritable := 'False'} : Bool;   // Auto Component 8
      ManSel8 { ExternalAccessible := 'False'; ExternalVisible := 'False'; ExternalWritable := 'False'} : Bool;   // Manu selected Component 8
      Man8 { ExternalAccessible := 'False'; ExternalVisible := 'False'; ExternalWritable := 'False'} : Bool;   // Manu Component 8
      AutoSel9 { ExternalAccessible := 'False'; ExternalVisible := 'False'; ExternalWritable := 'False'} : Bool;   // Auto selected Component 9
      Auto9 { ExternalAccessible := 'False'; ExternalVisible := 'False'; ExternalWritable := 'False'} : Bool;   // Auto Component 9
      ManSel9 { ExternalAccessible := 'False'; ExternalVisible := 'False'; ExternalWritable := 'False'} : Bool;   // Manu selected Component 9
      Man9 { ExternalAccessible := 'False'; ExternalVisible := 'False'; ExternalWritable := 'False'} : Bool;   // Manu Component 9
      AutoSel10 { ExternalAccessible := 'False'; ExternalVisible := 'False'; ExternalWritable := 'False'} : Bool;   // Auto selected Component 10
      Auto10 { ExternalAccessible := 'False'; ExternalVisible := 'False'; ExternalWritable := 'False'} : Bool;   // Auto Component 10
      ManSel10 { ExternalAccessible := 'False'; ExternalVisible := 'False'; ExternalWritable := 'False'} : Bool;   // Manu selected Component 10
      Man10 { ExternalAccessible := 'False'; ExternalVisible := 'False'; ExternalWritable := 'False'} : Bool;   // Manu Component 10
      AutoSel11 { ExternalAccessible := 'False'; ExternalVisible := 'False'; ExternalWritable := 'False'} : Bool;   // Auto selected Component 11
      Auto11 { ExternalAccessible := 'False'; ExternalVisible := 'False'; ExternalWritable := 'False'} : Bool;   // Auto Component 11
      ManSel11 { ExternalAccessible := 'False'; ExternalVisible := 'False'; ExternalWritable := 'False'} : Bool;   // Manu selected Component 11
      Man11 { ExternalAccessible := 'False'; ExternalVisible := 'False'; ExternalWritable := 'False'} : Bool;   // Manu Component 11
      AutoSel12 { ExternalAccessible := 'False'; ExternalVisible := 'False'; ExternalWritable := 'False'} : Bool;   // Auto selected Component 12
      Auto12 { ExternalAccessible := 'False'; ExternalVisible := 'False'; ExternalWritable := 'False'} : Bool;   // Auto Component 12
      ManSel12 { ExternalAccessible := 'False'; ExternalVisible := 'False'; ExternalWritable := 'False'} : Bool;   // Manu selected Component 12
      Man12 { ExternalAccessible := 'False'; ExternalVisible := 'False'; ExternalWritable := 'False'} : Bool;   // Manu Component 12
      AutoSel13 { ExternalAccessible := 'False'; ExternalVisible := 'False'; ExternalWritable := 'False'} : Bool;   // Auto selected Component 13
      Auto13 { ExternalAccessible := 'False'; ExternalVisible := 'False'; ExternalWritable := 'False'} : Bool;   // Auto Component 13
      ManSel13 { ExternalAccessible := 'False'; ExternalVisible := 'False'; ExternalWritable := 'False'} : Bool;   // Manu selected Component 13
      Man13 { ExternalAccessible := 'False'; ExternalVisible := 'False'; ExternalWritable := 'False'} : Bool;   // Manu Component 13
      AutoSel14 { ExternalAccessible := 'False'; ExternalVisible := 'False'; ExternalWritable := 'False'} : Bool;   // Auto selected Component 14
      Auto14 { ExternalAccessible := 'False'; ExternalVisible := 'False'; ExternalWritable := 'False'} : Bool;   // Auto Component 14
      ManSel14 { ExternalAccessible := 'False'; ExternalVisible := 'False'; ExternalWritable := 'False'} : Bool;   // Manu selected Component 14
      Man14 { ExternalAccessible := 'False'; ExternalVisible := 'False'; ExternalWritable := 'False'} : Bool;   // Manu Component 14
      AutoSel15 { ExternalAccessible := 'False'; ExternalVisible := 'False'; ExternalWritable := 'False'} : Bool;   // Auto selected Component 15
      Auto15 { ExternalAccessible := 'False'; ExternalVisible := 'False'; ExternalWritable := 'False'} : Bool;   // Auto Component 15
      ManSel15 { ExternalAccessible := 'False'; ExternalVisible := 'False'; ExternalWritable := 'False'} : Bool;   // Manu selected Component 15
      Man15 { ExternalAccessible := 'False'; ExternalVisible := 'False'; ExternalWritable := 'False'} : Bool;   // Manu Component 15
      AutoSel16 { ExternalAccessible := 'False'; ExternalVisible := 'False'; ExternalWritable := 'False'} : Bool;   // Auto selected Component 16
      Auto16 { ExternalAccessible := 'False'; ExternalVisible := 'False'; ExternalWritable := 'False'} : Bool;   // Auto Component 16
      ManSel16 { ExternalAccessible := 'False'; ExternalVisible := 'False'; ExternalWritable := 'False'} : Bool;   // Manu selected Component 16
      Man16 { ExternalAccessible := 'False'; ExternalVisible := 'False'; ExternalWritable := 'False'} : Bool;   // Manu Component 16
      AutoSel17 { ExternalAccessible := 'False'; ExternalVisible := 'False'; ExternalWritable := 'False'} : Bool;   // Auto selected Component 17
      Auto17 { ExternalAccessible := 'False'; ExternalVisible := 'False'; ExternalWritable := 'False'} : Bool;   // Auto Component 17
      ManSel17 { ExternalAccessible := 'False'; ExternalVisible := 'False'; ExternalWritable := 'False'} : Bool;   // Manu selected Component 17
      Man17 { ExternalAccessible := 'False'; ExternalVisible := 'False'; ExternalWritable := 'False'} : Bool;   // Manu Component 17
      AutoSel18 { ExternalAccessible := 'False'; ExternalVisible := 'False'; ExternalWritable := 'False'} : Bool;   // Auto selected Component 18
      Auto18 { ExternalAccessible := 'False'; ExternalVisible := 'False'; ExternalWritable := 'False'} : Bool;   // Auto Component 18
      ManSel18 { ExternalAccessible := 'False'; ExternalVisible := 'False'; ExternalWritable := 'False'} : Bool;   // Manu selected Component 18
      Man18 { ExternalAccessible := 'False'; ExternalVisible := 'False'; ExternalWritable := 'False'} : Bool;   // Manu Component 18
      AutoSel19 { ExternalAccessible := 'False'; ExternalVisible := 'False'; ExternalWritable := 'False'} : Bool;   // Auto selected Component 19
      Auto19 { ExternalAccessible := 'False'; ExternalVisible := 'False'; ExternalWritable := 'False'} : Bool;   // Auto Component 19
      ManSel19 { ExternalAccessible := 'False'; ExternalVisible := 'False'; ExternalWritable := 'False'} : Bool;   // Manu selected Component 19
      Man19 { ExternalAccessible := 'False'; ExternalVisible := 'False'; ExternalWritable := 'False'} : Bool;   // Manu Component 19
      AutoSel20 { ExternalAccessible := 'False'; ExternalVisible := 'False'; ExternalWritable := 'False'} : Bool;   // Auto selected Component 20
      Auto20 { ExternalAccessible := 'False'; ExternalVisible := 'False'; ExternalWritable := 'False'} : Bool;   // Auto Component 20
      ManSel20 { ExternalAccessible := 'False'; ExternalVisible := 'False'; ExternalWritable := 'False'} : Bool;   // Manu selected Component 20
      Man20 { ExternalAccessible := 'False'; ExternalVisible := 'False'; ExternalWritable := 'False'} : Bool;   // Manu Component 20
      Auto { ExternalAccessible := 'False'; ExternalVisible := 'False'; ExternalWritable := 'False'} : Bool;   // Auto Mode Summary
      Man { ExternalAccessible := 'False'; ExternalVisible := 'False'; ExternalWritable := 'False'} : Bool;   // Manual Mode Summary
      AutoSel { ExternalAccessible := 'False'; ExternalVisible := 'False'; ExternalWritable := 'False'} : Bool;   // Auto Mode Selected Summary
      ManSel { ExternalAccessible := 'False'; ExternalVisible := 'False'; ExternalWritable := 'False'} : Bool;   // Manual Mode Selected Summary
      TimerStartPBSel { ExternalAccessible := 'False'; ExternalVisible := 'False'; ExternalWritable := 'False'; S7_SetPoint := 'True'} : TOF_TIME;   // Timer
      TimerAlarmResetPBSel { ExternalAccessible := 'False'; ExternalVisible := 'False'; ExternalWritable := 'False'; S7_SetPoint := 'True'} : TOF_TIME;   // Timer
   END_VAR
BEGIN

REGION Network 1: **** 1 - Inputs **** Extract Mode Component 1
   // Extract Mode Component 1
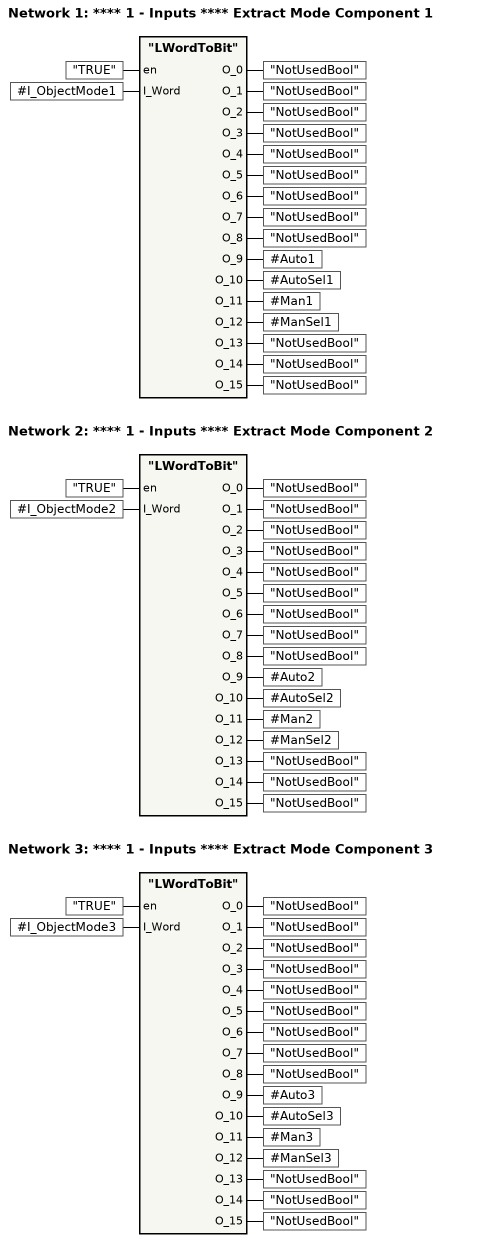
   IF "TRUE" THEN
       "LWordToBit"(I_Word := #I_ObjectMode1,
                    O_0 => "NotUsedBool",
                    O_1 => "NotUsedBool",
                    O_2 => "NotUsedBool",
                    O_3 => "NotUsedBool",
                    O_4 => "NotUsedBool",
                    O_5 => "NotUsedBool",
                    O_6 => "NotUsedBool",
                    O_7 => "NotUsedBool",
                    O_8 => "NotUsedBool",
                    O_9 => #Auto1,
                    O_10 => #AutoSel1,
                    O_11 => #Man1,
                    O_12 => #ManSel1,
                    O_13 => "NotUsedBool",
                    O_14 => "NotUsedBool",
                    O_15 => "NotUsedBool");
   END_IF;
END_REGION

REGION Network 2: **** 1 - Inputs **** Extract Mode Component 2
   // Extract Mode Component 2
   IF "TRUE" THEN
       "LWordToBit"(I_Word := #I_ObjectMode2,
                    O_0 => "NotUsedBool",
                    O_1 => "NotUsedBool",
                    O_2 => "NotUsedBool",
                    O_3 => "NotUsedBool",
                    O_4 => "NotUsedBool",
                    O_5 => "NotUsedBool",
                    O_6 => "NotUsedBool",
                    O_7 => "NotUsedBool",
                    O_8 => "NotUsedBool",
                    O_9 => #Auto2,
                    O_10 => #AutoSel2,
                    O_11 => #Man2,
                    O_12 => #ManSel2,
                    O_13 => "NotUsedBool",
                    O_14 => "NotUsedBool",
                    O_15 => "NotUsedBool");
   END_IF;
END_REGION

REGION Network 3: **** 1 - Inputs **** Extract Mode Component 3
   // Extract Mode Component 3
   IF "TRUE" THEN
       "LWordToBit"(I_Word := #I_ObjectMode3,
                    O_0 => "NotUsedBool",
                    O_1 => "NotUsedBool",
                    O_2 => "NotUsedBool",
                    O_3 => "NotUsedBool",
                    O_4 => "NotUsedBool",
                    O_5 => "NotUsedBool",
                    O_6 => "NotUsedBool",
                    O_7 => "NotUsedBool",
                    O_8 => "NotUsedBool",
                    O_9 => #Auto3,
                    O_10 => #AutoSel3,
                    O_11 => #Man3,
                    O_12 => #ManSel3,
                    O_13 => "NotUsedBool",
                    O_14 => "NotUsedBool",
                    O_15 => "NotUsedBool");
   END_IF;
END_REGION

REGION Network 4: **** 1 - Inputs **** Extract Mode Component 4
   // Extract Mode Component 4
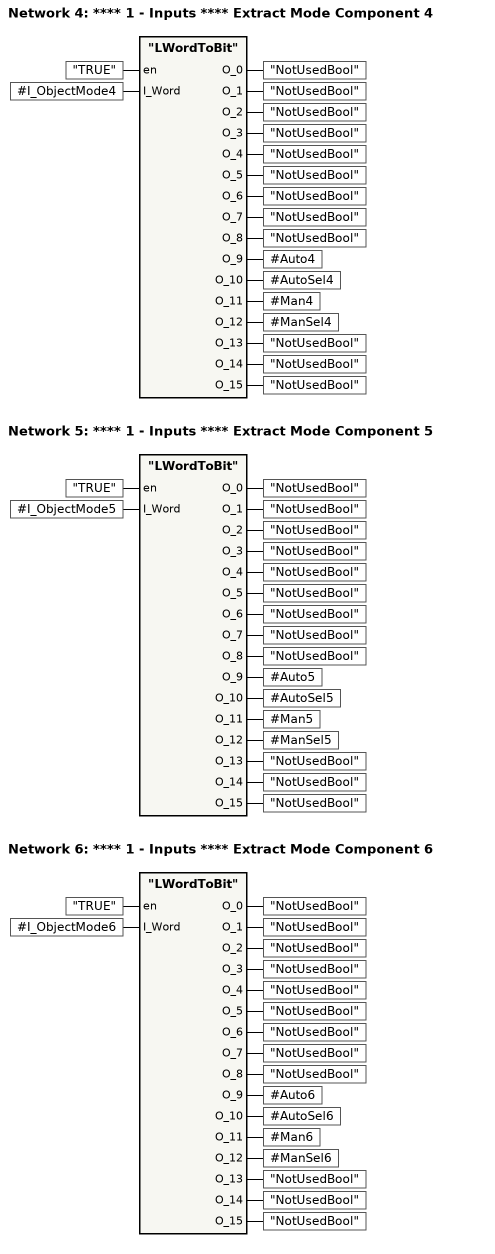
   IF "TRUE" THEN
       "LWordToBit"(I_Word := #I_ObjectMode4,
                    O_0 => "NotUsedBool",
                    O_1 => "NotUsedBool",
                    O_2 => "NotUsedBool",
                    O_3 => "NotUsedBool",
                    O_4 => "NotUsedBool",
                    O_5 => "NotUsedBool",
                    O_6 => "NotUsedBool",
                    O_7 => "NotUsedBool",
                    O_8 => "NotUsedBool",
                    O_9 => #Auto4,
                    O_10 => #AutoSel4,
                    O_11 => #Man4,
                    O_12 => #ManSel4,
                    O_13 => "NotUsedBool",
                    O_14 => "NotUsedBool",
                    O_15 => "NotUsedBool");
   END_IF;
END_REGION

REGION Network 5: **** 1 - Inputs **** Extract Mode Component 5
   // Extract Mode Component 5
   IF "TRUE" THEN
       "LWordToBit"(I_Word := #I_ObjectMode5,
                    O_0 => "NotUsedBool",
                    O_1 => "NotUsedBool",
                    O_2 => "NotUsedBool",
                    O_3 => "NotUsedBool",
                    O_4 => "NotUsedBool",
                    O_5 => "NotUsedBool",
                    O_6 => "NotUsedBool",
                    O_7 => "NotUsedBool",
                    O_8 => "NotUsedBool",
                    O_9 => #Auto5,
                    O_10 => #AutoSel5,
                    O_11 => #Man5,
                    O_12 => #ManSel5,
                    O_13 => "NotUsedBool",
                    O_14 => "NotUsedBool",
                    O_15 => "NotUsedBool");
   END_IF;
END_REGION

REGION Network 6: **** 1 - Inputs **** Extract Mode Component 6
   // Extract Mode Component 6
   IF "TRUE" THEN
       "LWordToBit"(I_Word := #I_ObjectMode6,
                    O_0 => "NotUsedBool",
                    O_1 => "NotUsedBool",
                    O_2 => "NotUsedBool",
                    O_3 => "NotUsedBool",
                    O_4 => "NotUsedBool",
                    O_5 => "NotUsedBool",
                    O_6 => "NotUsedBool",
                    O_7 => "NotUsedBool",
                    O_8 => "NotUsedBool",
                    O_9 => #Auto6,
                    O_10 => #AutoSel6,
                    O_11 => #Man6,
                    O_12 => #ManSel6,
                    O_13 => "NotUsedBool",
                    O_14 => "NotUsedBool",
                    O_15 => "NotUsedBool");
   END_IF;
END_REGION

REGION Network 7: **** 1 - Inputs **** Extract Mode Component 7
   // Extract Mode Component 7
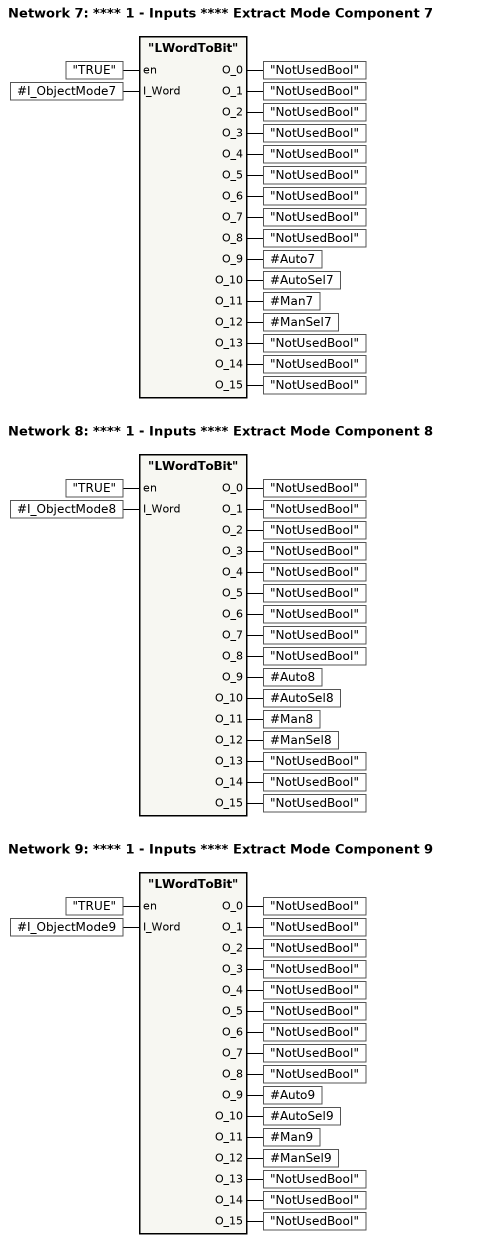
   IF "TRUE" THEN
       "LWordToBit"(I_Word := #I_ObjectMode7,
                    O_0 => "NotUsedBool",
                    O_1 => "NotUsedBool",
                    O_2 => "NotUsedBool",
                    O_3 => "NotUsedBool",
                    O_4 => "NotUsedBool",
                    O_5 => "NotUsedBool",
                    O_6 => "NotUsedBool",
                    O_7 => "NotUsedBool",
                    O_8 => "NotUsedBool",
                    O_9 => #Auto7,
                    O_10 => #AutoSel7,
                    O_11 => #Man7,
                    O_12 => #ManSel7,
                    O_13 => "NotUsedBool",
                    O_14 => "NotUsedBool",
                    O_15 => "NotUsedBool");
   END_IF;
END_REGION

REGION Network 8: **** 1 - Inputs **** Extract Mode Component 8
   // Extract Mode Component 8
   IF "TRUE" THEN
       "LWordToBit"(I_Word := #I_ObjectMode8,
                    O_0 => "NotUsedBool",
                    O_1 => "NotUsedBool",
                    O_2 => "NotUsedBool",
                    O_3 => "NotUsedBool",
                    O_4 => "NotUsedBool",
                    O_5 => "NotUsedBool",
                    O_6 => "NotUsedBool",
                    O_7 => "NotUsedBool",
                    O_8 => "NotUsedBool",
                    O_9 => #Auto8,
                    O_10 => #AutoSel8,
                    O_11 => #Man8,
                    O_12 => #ManSel8,
                    O_13 => "NotUsedBool",
                    O_14 => "NotUsedBool",
                    O_15 => "NotUsedBool");
   END_IF;
END_REGION

REGION Network 9: **** 1 - Inputs **** Extract Mode Component 9
   // Extract Mode Component 9
   IF "TRUE" THEN
       "LWordToBit"(I_Word := #I_ObjectMode9,
                    O_0 => "NotUsedBool",
                    O_1 => "NotUsedBool",
                    O_2 => "NotUsedBool",
                    O_3 => "NotUsedBool",
                    O_4 => "NotUsedBool",
                    O_5 => "NotUsedBool",
                    O_6 => "NotUsedBool",
                    O_7 => "NotUsedBool",
                    O_8 => "NotUsedBool",
                    O_9 => #Auto9,
                    O_10 => #AutoSel9,
                    O_11 => #Man9,
                    O_12 => #ManSel9,
                    O_13 => "NotUsedBool",
                    O_14 => "NotUsedBool",
                    O_15 => "NotUsedBool");
   END_IF;
END_REGION

REGION Network 10: **** 1 - Inputs **** Extract Mode Component 10
   // Extract Mode Component 10
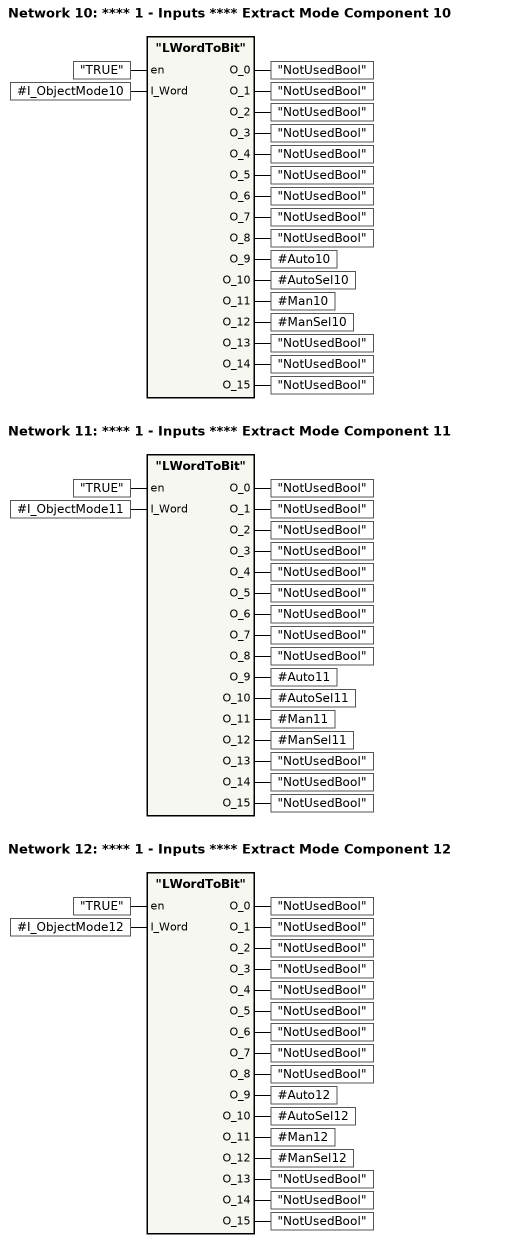
   IF "TRUE" THEN
       "LWordToBit"(I_Word := #I_ObjectMode10,
                    O_0 => "NotUsedBool",
                    O_1 => "NotUsedBool",
                    O_2 => "NotUsedBool",
                    O_3 => "NotUsedBool",
                    O_4 => "NotUsedBool",
                    O_5 => "NotUsedBool",
                    O_6 => "NotUsedBool",
                    O_7 => "NotUsedBool",
                    O_8 => "NotUsedBool",
                    O_9 => #Auto10,
                    O_10 => #AutoSel10,
                    O_11 => #Man10,
                    O_12 => #ManSel10,
                    O_13 => "NotUsedBool",
                    O_14 => "NotUsedBool",
                    O_15 => "NotUsedBool");
   END_IF;
END_REGION

REGION Network 11: **** 1 - Inputs **** Extract Mode Component 11
   // Extract Mode Component 11
   IF "TRUE" THEN
       "LWordToBit"(I_Word := #I_ObjectMode11,
                    O_0 => "NotUsedBool",
                    O_1 => "NotUsedBool",
                    O_2 => "NotUsedBool",
                    O_3 => "NotUsedBool",
                    O_4 => "NotUsedBool",
                    O_5 => "NotUsedBool",
                    O_6 => "NotUsedBool",
                    O_7 => "NotUsedBool",
                    O_8 => "NotUsedBool",
                    O_9 => #Auto11,
                    O_10 => #AutoSel11,
                    O_11 => #Man11,
                    O_12 => #ManSel11,
                    O_13 => "NotUsedBool",
                    O_14 => "NotUsedBool",
                    O_15 => "NotUsedBool");
   END_IF;
END_REGION

REGION Network 12: **** 1 - Inputs **** Extract Mode Component 12
   // Extract Mode Component 12
   IF "TRUE" THEN
       "LWordToBit"(I_Word := #I_ObjectMode12,
                    O_0 => "NotUsedBool",
                    O_1 => "NotUsedBool",
                    O_2 => "NotUsedBool",
                    O_3 => "NotUsedBool",
                    O_4 => "NotUsedBool",
                    O_5 => "NotUsedBool",
                    O_6 => "NotUsedBool",
                    O_7 => "NotUsedBool",
                    O_8 => "NotUsedBool",
                    O_9 => #Auto12,
                    O_10 => #AutoSel12,
                    O_11 => #Man12,
                    O_12 => #ManSel12,
                    O_13 => "NotUsedBool",
                    O_14 => "NotUsedBool",
                    O_15 => "NotUsedBool");
   END_IF;
END_REGION

REGION Network 13: **** 1 - Inputs **** Extract Mode Component 13
   // Extract Mode Component 13
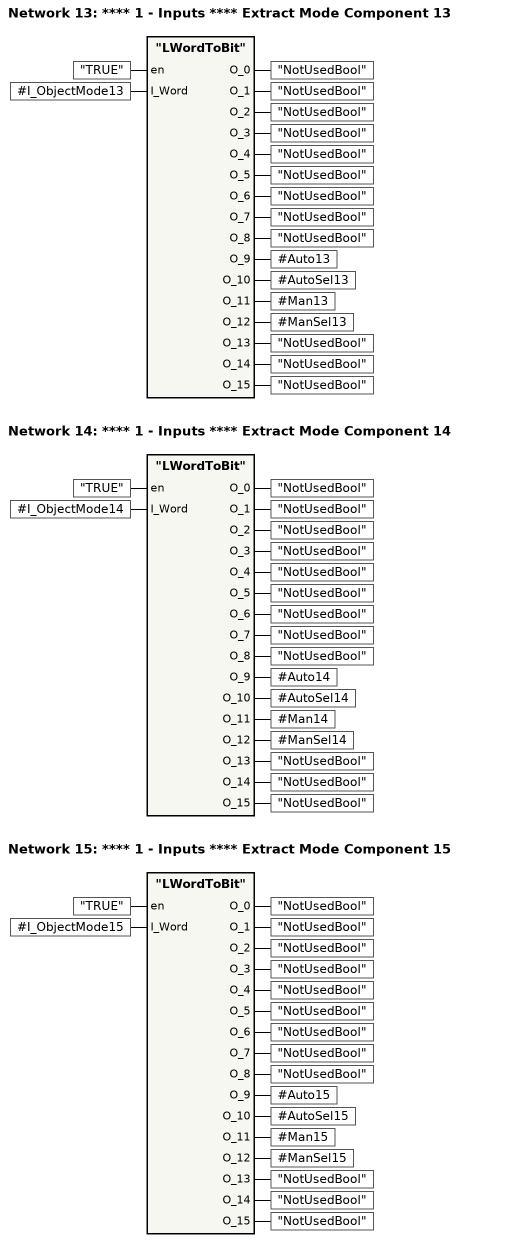
   IF "TRUE" THEN
       "LWordToBit"(I_Word := #I_ObjectMode13,
                    O_0 => "NotUsedBool",
                    O_1 => "NotUsedBool",
                    O_2 => "NotUsedBool",
                    O_3 => "NotUsedBool",
                    O_4 => "NotUsedBool",
                    O_5 => "NotUsedBool",
                    O_6 => "NotUsedBool",
                    O_7 => "NotUsedBool",
                    O_8 => "NotUsedBool",
                    O_9 => #Auto13,
                    O_10 => #AutoSel13,
                    O_11 => #Man13,
                    O_12 => #ManSel13,
                    O_13 => "NotUsedBool",
                    O_14 => "NotUsedBool",
                    O_15 => "NotUsedBool");
   END_IF;
END_REGION

REGION Network 14: **** 1 - Inputs **** Extract Mode Component 14
   // Extract Mode Component 14
   IF "TRUE" THEN
       "LWordToBit"(I_Word := #I_ObjectMode14,
                    O_0 => "NotUsedBool",
                    O_1 => "NotUsedBool",
                    O_2 => "NotUsedBool",
                    O_3 => "NotUsedBool",
                    O_4 => "NotUsedBool",
                    O_5 => "NotUsedBool",
                    O_6 => "NotUsedBool",
                    O_7 => "NotUsedBool",
                    O_8 => "NotUsedBool",
                    O_9 => #Auto14,
                    O_10 => #AutoSel14,
                    O_11 => #Man14,
                    O_12 => #ManSel14,
                    O_13 => "NotUsedBool",
                    O_14 => "NotUsedBool",
                    O_15 => "NotUsedBool");
   END_IF;
END_REGION

REGION Network 15: **** 1 - Inputs **** Extract Mode Component 15
   // Extract Mode Component 15
   IF "TRUE" THEN
       "LWordToBit"(I_Word := #I_ObjectMode15,
                    O_0 => "NotUsedBool",
                    O_1 => "NotUsedBool",
                    O_2 => "NotUsedBool",
                    O_3 => "NotUsedBool",
                    O_4 => "NotUsedBool",
                    O_5 => "NotUsedBool",
                    O_6 => "NotUsedBool",
                    O_7 => "NotUsedBool",
                    O_8 => "NotUsedBool",
                    O_9 => #Auto15,
                    O_10 => #AutoSel15,
                    O_11 => #Man15,
                    O_12 => #ManSel15,
                    O_13 => "NotUsedBool",
                    O_14 => "NotUsedBool",
                    O_15 => "NotUsedBool");
   END_IF;
END_REGION

REGION Network 16: **** 1 - Inputs **** Extract Mode Component 16
   // Extract Mode Component 16
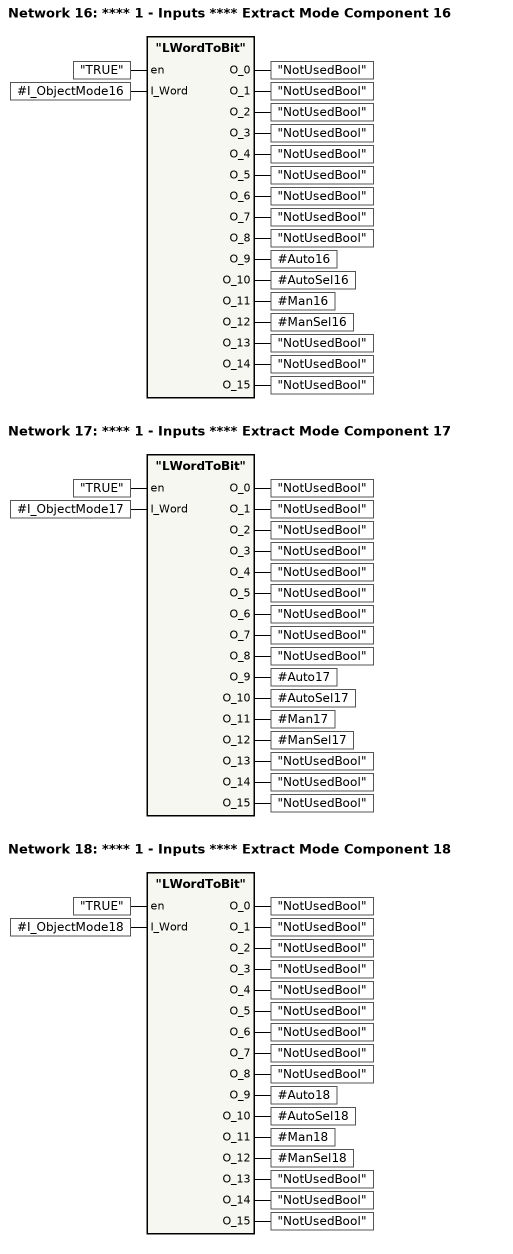
   IF "TRUE" THEN
       "LWordToBit"(I_Word := #I_ObjectMode16,
                    O_0 => "NotUsedBool",
                    O_1 => "NotUsedBool",
                    O_2 => "NotUsedBool",
                    O_3 => "NotUsedBool",
                    O_4 => "NotUsedBool",
                    O_5 => "NotUsedBool",
                    O_6 => "NotUsedBool",
                    O_7 => "NotUsedBool",
                    O_8 => "NotUsedBool",
                    O_9 => #Auto16,
                    O_10 => #AutoSel16,
                    O_11 => #Man16,
                    O_12 => #ManSel16,
                    O_13 => "NotUsedBool",
                    O_14 => "NotUsedBool",
                    O_15 => "NotUsedBool");
   END_IF;
END_REGION

REGION Network 17: **** 1 - Inputs **** Extract Mode Component 17
   // Extract Mode Component 17
   IF "TRUE" THEN
       "LWordToBit"(I_Word := #I_ObjectMode17,
                    O_0 => "NotUsedBool",
                    O_1 => "NotUsedBool",
                    O_2 => "NotUsedBool",
                    O_3 => "NotUsedBool",
                    O_4 => "NotUsedBool",
                    O_5 => "NotUsedBool",
                    O_6 => "NotUsedBool",
                    O_7 => "NotUsedBool",
                    O_8 => "NotUsedBool",
                    O_9 => #Auto17,
                    O_10 => #AutoSel17,
                    O_11 => #Man17,
                    O_12 => #ManSel17,
                    O_13 => "NotUsedBool",
                    O_14 => "NotUsedBool",
                    O_15 => "NotUsedBool");
   END_IF;
END_REGION

REGION Network 18: **** 1 - Inputs **** Extract Mode Component 18
   // Extract Mode Component 18
   IF "TRUE" THEN
       "LWordToBit"(I_Word := #I_ObjectMode18,
                    O_0 => "NotUsedBool",
                    O_1 => "NotUsedBool",
                    O_2 => "NotUsedBool",
                    O_3 => "NotUsedBool",
                    O_4 => "NotUsedBool",
                    O_5 => "NotUsedBool",
                    O_6 => "NotUsedBool",
                    O_7 => "NotUsedBool",
                    O_8 => "NotUsedBool",
                    O_9 => #Auto18,
                    O_10 => #AutoSel18,
                    O_11 => #Man18,
                    O_12 => #ManSel18,
                    O_13 => "NotUsedBool",
                    O_14 => "NotUsedBool",
                    O_15 => "NotUsedBool");
   END_IF;
END_REGION

REGION Network 19: **** 1 - Inputs **** Extract Mode Component 19
   // Extract Mode Component 19
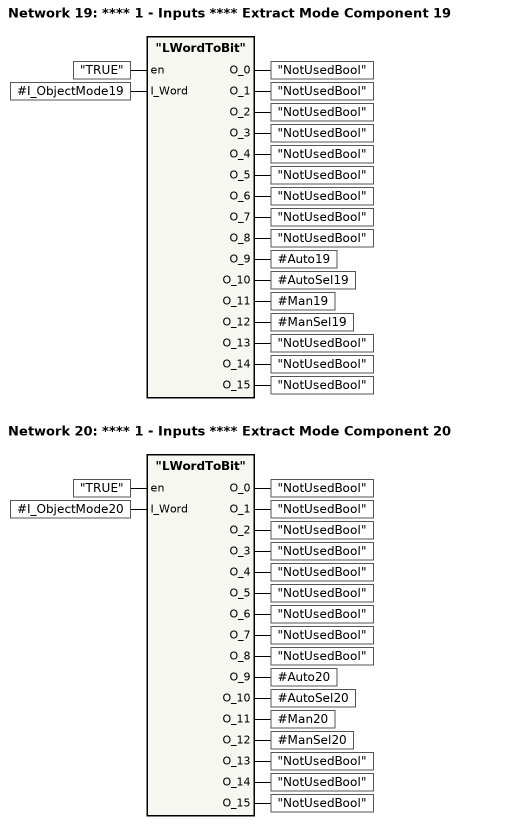
   IF "TRUE" THEN
       "LWordToBit"(I_Word := #I_ObjectMode19,
                    O_0 => "NotUsedBool",
                    O_1 => "NotUsedBool",
                    O_2 => "NotUsedBool",
                    O_3 => "NotUsedBool",
                    O_4 => "NotUsedBool",
                    O_5 => "NotUsedBool",
                    O_6 => "NotUsedBool",
                    O_7 => "NotUsedBool",
                    O_8 => "NotUsedBool",
                    O_9 => #Auto19,
                    O_10 => #AutoSel19,
                    O_11 => #Man19,
                    O_12 => #ManSel19,
                    O_13 => "NotUsedBool",
                    O_14 => "NotUsedBool",
                    O_15 => "NotUsedBool");
   END_IF;
END_REGION

REGION Network 20: **** 1 - Inputs **** Extract Mode Component 20
   // Extract Mode Component 20
   IF "TRUE" THEN
       "LWordToBit"(I_Word := #I_ObjectMode20,
                    O_0 => "NotUsedBool",
                    O_1 => "NotUsedBool",
                    O_2 => "NotUsedBool",
                    O_3 => "NotUsedBool",
                    O_4 => "NotUsedBool",
                    O_5 => "NotUsedBool",
                    O_6 => "NotUsedBool",
                    O_7 => "NotUsedBool",
                    O_8 => "NotUsedBool",
                    O_9 => #Auto20,
                    O_10 => #AutoSel20,
                    O_11 => #Man20,
                    O_12 => #ManSel20,
                    O_13 => "NotUsedBool",
                    O_14 => "NotUsedBool",
                    O_15 => "NotUsedBool");
   END_IF;
END_REGION

REGION Network 21: **** 4.6 - Machine status - Indications **** Summary Auto Mode
   // Summary Auto Mode
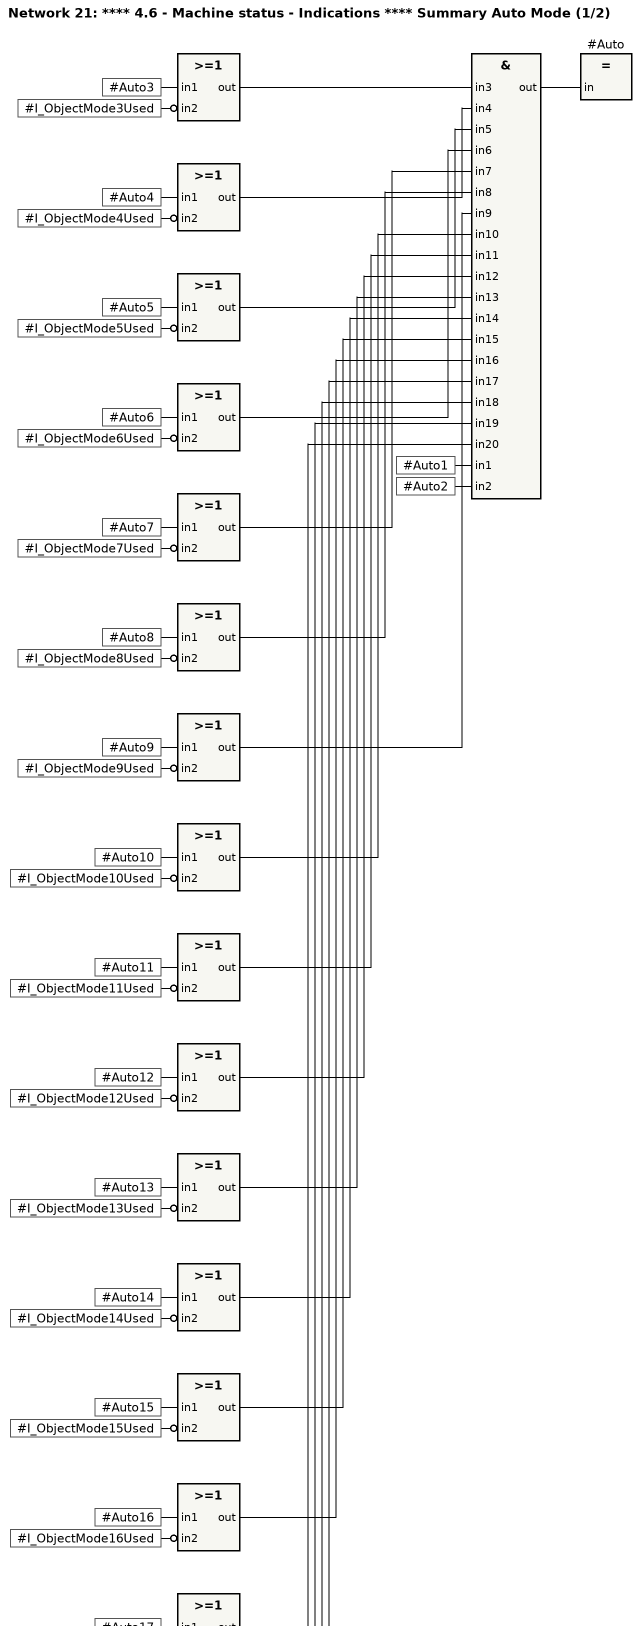
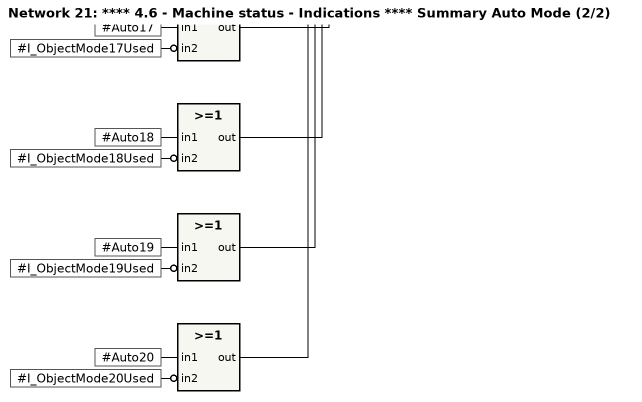
   #Auto := (#Auto3 OR NOT #I_ObjectMode3Used) AND (#Auto4 OR NOT #I_ObjectMode4Used) AND (#Auto5 OR NOT #I_ObjectMode5Used) AND (#Auto6 OR NOT #I_ObjectMode6Used) AND (#Auto7 OR NOT #I_ObjectMode7Used) AND (#Auto8 OR NOT #I_ObjectMode8Used) AND (#Auto9 OR NOT #I_ObjectMode9Used) AND (#Auto10 OR NOT #I_ObjectMode10Used) AND (#Auto11 OR NOT #I_ObjectMode11Used) AND (#Auto12 OR NOT #I_ObjectMode12Used) AND (#Auto13 OR NOT #I_ObjectMode13Used) AND (#Auto14 OR NOT #I_ObjectMode14Used) AND (#Auto15 OR NOT #I_ObjectMode15Used) AND (#Auto16 OR NOT #I_ObjectMode16Used) AND (#Auto17 OR NOT #I_ObjectMode17Used) AND (#Auto18 OR NOT #I_ObjectMode18Used) AND (#Auto19 OR NOT #I_ObjectMode19Used) AND (#Auto20 OR NOT #I_ObjectMode20Used) AND #Auto1 AND #Auto2;
END_REGION

REGION Network 22: **** 4.6 - Machine status - Indications **** Summary AutoSel
   // Summary AutoSel
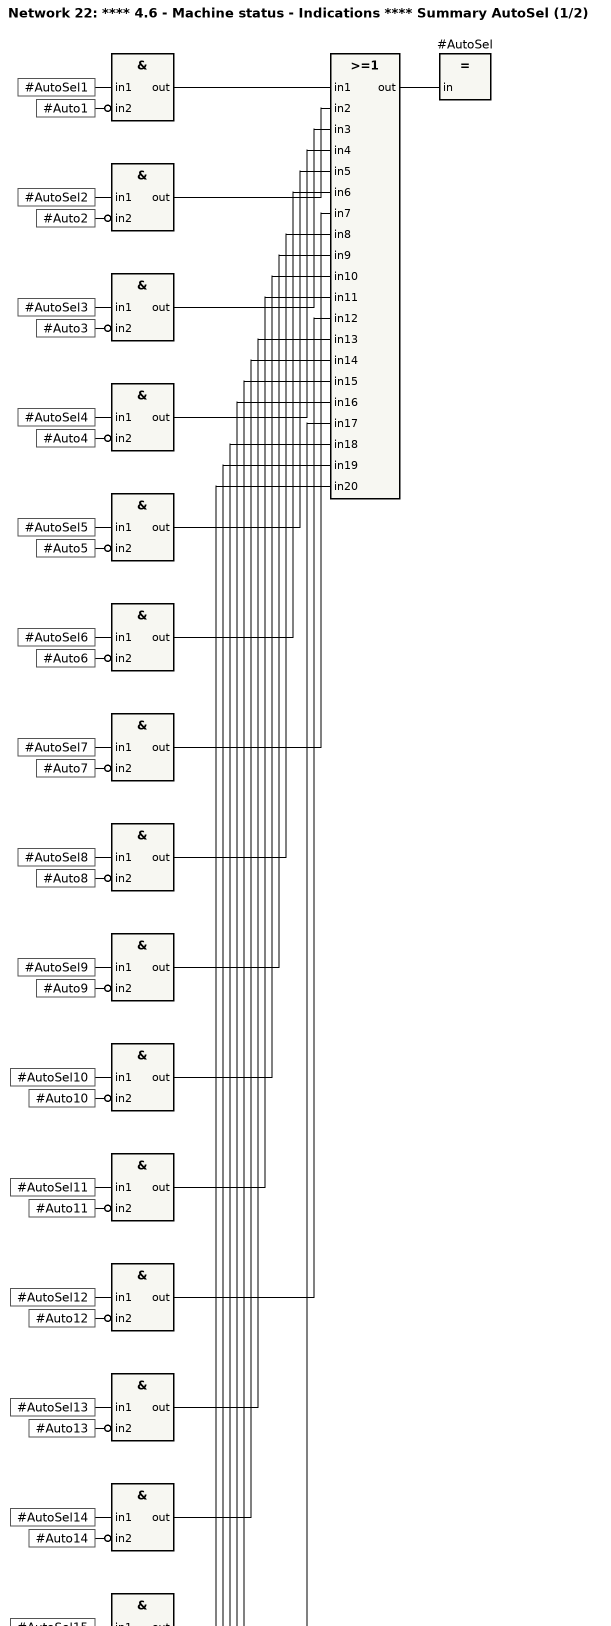
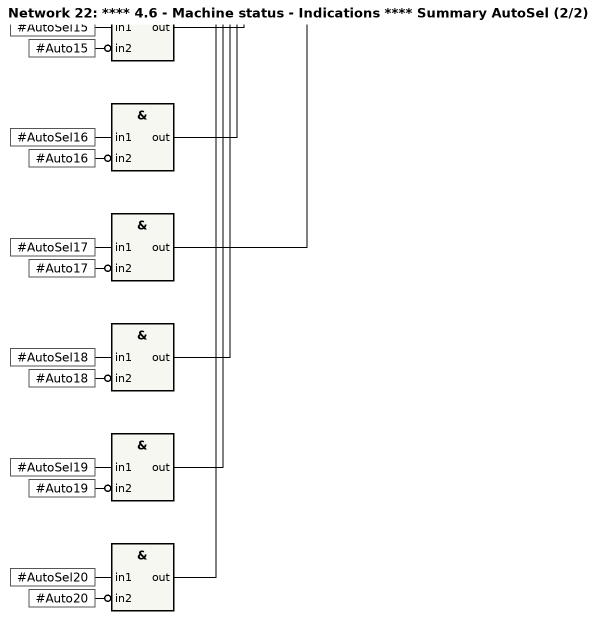
   #AutoSel := (#AutoSel1 AND NOT #Auto1) OR (#AutoSel2 AND NOT #Auto2) OR (#AutoSel3 AND NOT #Auto3) OR (#AutoSel4 AND NOT #Auto4) OR (#AutoSel5 AND NOT #Auto5) OR (#AutoSel6 AND NOT #Auto6) OR (#AutoSel7 AND NOT #Auto7) OR (#AutoSel8 AND NOT #Auto8) OR (#AutoSel9 AND NOT #Auto9) OR (#AutoSel10 AND NOT #Auto10) OR (#AutoSel11 AND NOT #Auto11) OR (#AutoSel12 AND NOT #Auto12) OR (#AutoSel13 AND NOT #Auto13) OR (#AutoSel14 AND NOT #Auto14) OR (#AutoSel15 AND NOT #Auto15) OR (#AutoSel16 AND NOT #Auto16) OR (#AutoSel17 AND NOT #Auto17) OR (#AutoSel18 AND NOT #Auto18) OR (#AutoSel19 AND NOT #Auto19) OR (#AutoSel20 AND NOT #Auto20);
END_REGION

REGION Network 23: **** 4.6 - Machine status - Indications **** Summary AutoSel
   // Summary AutoSel
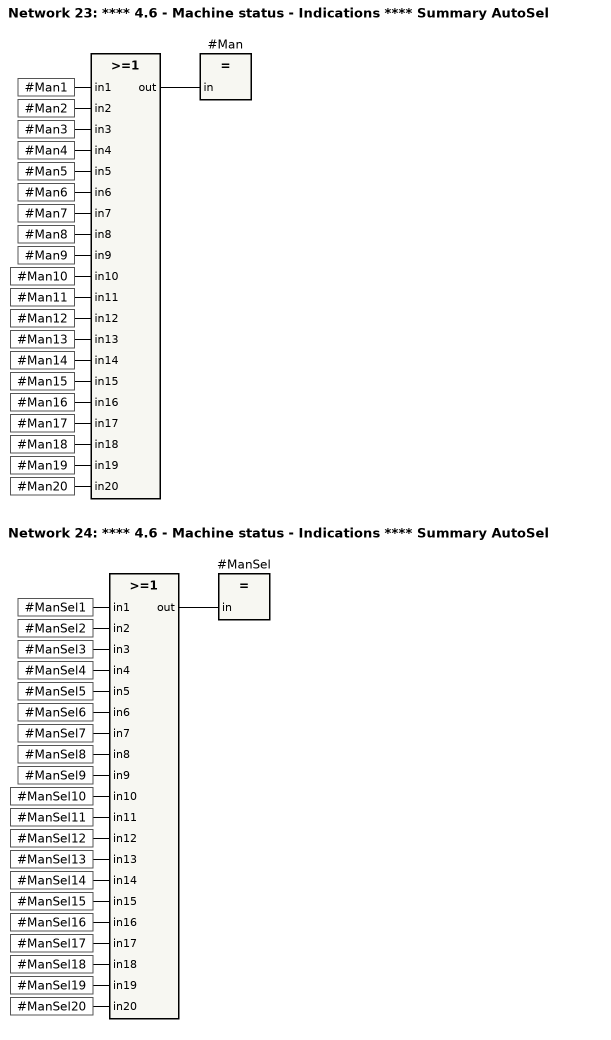
   #Man := #Man1 OR #Man2 OR #Man3 OR #Man4 OR #Man5 OR #Man6 OR #Man7 OR #Man8 OR #Man9 OR #Man10 OR #Man11 OR #Man12 OR #Man13 OR #Man14 OR #Man15 OR #Man16 OR #Man17 OR #Man18 OR #Man19 OR #Man20;
END_REGION

REGION Network 24: **** 4.6 - Machine status - Indications **** Summary AutoSel
   // Summary AutoSel
   #ManSel := #ManSel1 OR #ManSel2 OR #ManSel3 OR #ManSel4 OR #ManSel5 OR #ManSel6 OR #ManSel7 OR #ManSel8 OR #ManSel9 OR #ManSel10 OR #ManSel11 OR #ManSel12 OR #ManSel13 OR #ManSel14 OR #ManSel15 OR #ManSel16 OR #ManSel17 OR #ManSel18 OR #ManSel19 OR #ManSel20;
END_REGION

REGION Network 25: **** 4.6 - Machine Status - Indications **** Animation
   // Animation
